(* CoDeSys 2.3.9.50 project: Indo_Tex.pro *)
(* Libraries: COMlibV2.lib 24.2.14 12:45:46, FB_DateTime.lib 15.2.16 16:36:26, TcMath.lib 23.9.04 14:15:30, SysLibVisu.lib 7.7.04 17:17:22, SysLibTargetVisu.lib 16.6.08 15:24:26, TcEtherCAT.lib 30.11.16 18:52:18, TcUtilities.lib 3.2.16 15:08:58, TcSystem.lib 7.6.16 10:01:22, TcBaseMath.lib 27.7.04 11:07:56, STANDARD.LIB 5.6.98 11:03:02, TcBase.lib 14.5.09 11:14:08, ModbusRTU.lib 19.12.16 16:50:06, TcSystemCX.lib 7.9.16 11:51:26 *)

(* Global variable list: Date_Time *)
VAR_GLOBAL
	FB_DateTime_1: FB_DateTime;
	sHourPreFix: STRING;
	sHou: STRING;
	sDayPreFix: STRING;
	sDay: STRING;
	sMonthPreFix: STRING;
	sMonth: STRING;
	sDayF: STRING;
	sMonthF: STRING;
	sDayMonth: STRING;
	sDayMonthYear: STRING;
	sDaateReport: STRING;
	sDayMonthYear1: STRING;

END_VAR

(* Global variable list: GVL_Alarm *)
VAR_GLOBAL
	RS_Error_1: RS_Error;
	RS_Error_2: RS_Error;
	RS_Error_3: RS_Error;
	RS_Error_4: RS_Error;
	RS_Error_5: RS_Error;
	RS_Error_6: RS_Error;
	RS_Error_7: RS_Error;

	bASealConvEnd1: BOOL;
	AlarmMess2: STRING(80);
	AlarmMess1: STRING(80);
	AlarWrap: STRING(80);
	CountMess: STRING(80);
	AlarmMessg: STRING(80);
	UnitASenSelet: UINT;
	SealingStep: INT;
	AlarmWrpConyMess: STRING(80);
	ConeMissAlarm: STRING(80);

	bAConeFeedCylRsError: BOOL;
	bAFwdCylRsError: BOOL;
	bAWrappingCylRsError: BOOL;
	bAWrappingCylRs1Error: BOOL;
	bAWrappingCylRs2Error: BOOL;
	bAWrappingCylRs3Error: BOOL;
	bAWrapCylRsErrorAuto: BOOL;
	bAError: BOOL;
	bASealTopCylRsError: BOOL;
	bASealBotCylRsError: BOOL;
	bASealTopBotCylRsError: BOOL;
	bASealSepXCylRsError: BOOL;
	bASealSepYCylRsError: BOOL;
	bASupplyPressureError: BOOL;
	HmiSupplyPressureMsg: STRING;
	bAFilmNotloaded: BOOL;
	bAConeMissAtSealConv: BOOL;
	bAEmergencyPressed: BOOL;
	bEmPopUp: BOOL;
	bAConeMissErrorAtWrpConv: BOOL;
	ConeAlignErr: BOOL;
	ConeMissAlarm1: STRING;
	ConeMissAlarm2: STRING;
	bAFlimNotLoaded: BOOL;
	bAPolythinSheetError: BOOL;
	bFilmErrClear: BOOL;
	bASepYAxisRsErrorChkBit: BOOL;
	bASepYAxisRsErrorChkBit1: BOOL;
	bABuzzer: BOOL;
	PressureChkTimer: TON;
	bAStop: BOOL;

	bAErrorChkBit: BOOL;
	bCheckWrappingSen: BOOL;
	bPloySheetSensError: BOOL;
	checkPolySheet2: BOOL;
	bAErrorChkBit2: BOOL;
	bCheckWrappingSen2: BOOL;
	bAErrorChkBit3: BOOL;
	bCheckWrappingSen3: BOOL;
	bWrapConvStopped2Temp: BOOL;
	SealingOk: BOOL;
	CycleComplete: BOOL;
	CycleComplete1: BOOL;
	SGrossWtNokMsg: STRING;

	SGrossWtCylEndSenErrMsg: STRING;
	bGrossWtCylEndSenError: BOOL;
END_VAR

(* Global variable list: GVL_Auto *)
VAR_GLOBAL
	bAutoModeOn: BOOL;
	bAPauseSeq: BOOL;
	bUnitBRowStopperStarted: BOOL;
	bUnitARowStopperStarted: BOOL;
	bAUnitAWeighOk: BOOL;
	bAConeFeedOver: BOOL;
	bAWrappingConvStart3: BOOL;
	bAWrappingConvStart1: BOOL;
	bAWrappingConvStart2: BOOL;
			bA3ConeWrappOver: BOOL;
	bA4thWrappOver: BOOL;
	bA6thConeWrappOver: BOOL;
	bA8thConeWrappOver: BOOL;
	bA6ConeWrappOver23: BOOL;
	AlarmMess: STRING(80);
	bAWrappingCone123OnAuto: BOOL;
	bAFwdPistonComp1: BOOL;
	bAFwdPistonComp2: BOOL;
	bAFwdPistonComp3: BOOL;
	bAConvFirstStart: BOOL;
	UnitACompleteCheckCount: CTU;
	bRetUnitAStart: BOOL;
	bRetUnitBStart: BOOL;
	bAUnitBWeighOk: BOOL;
	ConeInCompleteB: BOOL;
	(*UnitAConeCompChkCount: CTU;*)
	iSensorOnVal: USINT;
	bFwdPistonStartTemp: BOOL;
	bConeMiss1AtWrapConv: BOOL;
	bConeMiss2tWrapConv: BOOL;
	bConeMiss2AtWrapConv: BOOL;
	ConeMissbit: BOOL;
	CTU_1: CTU;
	bAPauseEnable: BOOL;
	SealComDlyTemp: TIME;
	bAMcStartInAuto: BOOL;
	bPauseExtend: BOOL;
	bAutoModeOff: BOOL;
	iTotalNoOfCones: BOOL;
	iATotalNoOfCones: INT;
	bAMcReady: BOOL;
	bAMcRunninig: BOOL;
	bAFilmLoaded: BOOL;
	bAWrapConStart: BOOL;
	bA3ConeWrappOverTemp: BOOL;
	bABypassOn: BOOL;
	bIntialAckBit: BOOL;
	ConeInComplete: BOOL;
	ConeInCompletetest: BOOL;
	ConeInCompleteTestbitB: BOOL;
	bUnitACounterDIsable: BOOL;
	ConeInCompleteA: BOOL;
	bAOneMinConvStart: BOOL;
	bAWrapwait: BOOL;
END_VAR

(* Global variable list: GVL_Hmi *)
VAR_GLOBAL
	bStopHmi: BOOL;
	bInitializeHmi: BOOL;

	HMIFeedPiston: STRING(80);
	HMIWrapPiston1: STRING(80);
	HMIWrapPiston2: STRING(80);
	HMIWrapPiston3: STRING(80);
	HMIForwdPiston:STRING(80);
	HMISealBotPiston:STRING(80);
	HMISealTopPiston:STRING(80);
	HmiXAxisPiston:STRING(80);
	HmiYAxisPiston:STRING(80);
	bErrorReset: BOOL;
	bPauseHmi: BOOL;
	bResumeHmi: BOOL;
	bResetTemp: BOOL;
	bHmiAck: BOOL;

	b18ConeModelHmi: BOOL;
	b12ConeModelHmi:BOOL;
	b24ConeModelHmi: BOOL;
	b32ConeModelHmi: BOOL;
	sAMcModeStatus: STRING;
	bAUnitBConeCrossed: BOOL;
	bAInializeStarted: BOOL;
	PopUp: BOOL;
	sAlarmStatus: STRING;
	bNegTolDisableHMI: BOOL;
	bNegTolEnableHMI: BOOL;
	bPrssurePopUp: BOOL;
	UnitAConeCountHMI: INT;
	UnitAConeCountHMI_1: INT;
	UnitBConeCountHMI: INT;
	b16ConeModelHmi: BOOL;
	WrapConeSenDetMes: STRING;
	bAmberbit2: BOOL;
	Pgm_NoHmi: INT;
	FileCreateTemp: BOOL;
	bACyclePass: BOOL;
	iCartoNoHmi: STRING;
	(*iLotNoHmi: STRING;*)
	var_1: REAL;
	var_5: REAL;
	LogYear: STRING;
	LogMonth: STRING;
	logDay: STRING;
	sTIME: STRING;
	sDATEFinal: STRING;
	DateTimeVar: STRING;
	wTodayToHmi: STRING;
	bInterlockInitial_2: BOOL;
	sMessage: STRING;
	bReadGWieght: BOOL;
	bAReset_all_error: BOOL;



	(*ProgramNoHmi:INT;
	CountCodeHmi:STRING;
	CartonNoHmi:INT;
	DefaultNetWeightHmi:REAL;
	DefaultGrossWeightHmi:REAL;
	BlendHmi:STRING;
	ShadeHmi:STRING;
	ConeTipHmi:STRING;
	ConeNettHmi:STRING;
	ConeLengthHmi:REAL;
	Cones:INT;
	Dom_ExpHmi:STRING;
	PackTypeHmi:STRING;*)




	LotASelected: BOOL;
	LotACartonNo: INT;
	LotBSelected: BOOL;
	LotBCartonNo: INT;
	LotCSelected: BOOL;
	LotDSelected: BOOL;
	LotESelected: BOOL;
	LotFSelected: BOOL;
	LotCCartonNo: INT;
	LotDCartonNo:  INT;
	LotECartonNo:  INT;
	LotFCartonNo: INT;
	LotA: INT;

	LotB: INT;

	LotC: INT;

	LotAHmi: BOOL;
	LotBHmi: BOOL;
	LotCHmi: BOOL;
	CurrentCartonNo:INT;
	LotNoChange: BOOL;
	ParametesSave: BOOL;
END_VAR

VAR_GLOBAL RETAIN
(*VAR_GLOBAL PERSISTENT*)
	b12ConeModelSelected AT %Q*: BOOL;
	b18ConeModelSelected AT %Q*: BOOL;
	b24ConeModelSelected AT %Q*: BOOL;
	b32ConeModelSelected AT %Q*: BOOL;
	rSealCompDlyHmi AT %Q*: REAL;
	iNetTolHmi AT %Q*: REAL;
	iNetWtHmi AT %Q*: REAL;
	iLotNoHmi AT %Q*: STRING;
	iWorkOrderNoHmi AT %Q*:STRING;
	NegToleranceEnabled AT %Q*: BOOL;
	b16ConeModelSelected AT %Q*: BOOL;

	ProgramNoHmi AT %Q*: INT;
	CountCodeHmi AT %Q*: STRING(80);
	CartonNoHmi AT %Q*: INT;
	DefaultNetWeightHmi AT %Q*: REAL;
	DefaultGrossWeightHmi AT %Q*: REAL;
	EmptyConeWt AT %Q*: REAL;
	BlendHmi AT %Q*: STRING(80);
	ShadeHmi AT %Q*: STRING(80);
	ConeTipHmi AT %Q*: STRING(80);
	ConeNettHmi AT %Q*: STRING(80);
	ConeLengthHmi AT %Q*: REAL;
	Cones:INT;
	Dom_ExpHmi AT %Q*: STRING(80);
	PackTypeHmi AT %Q*: STRING(80);
	ItemCodeHmi AT %Q*: STRING(80);
	IssueDesp AT %Q*: STRING(80);
	Location AT %Q*: STRING(80);
	Description AT %Q*: STRING(80);
	Remarks AT %Q*: STRING(80);
	Fyear AT %Q*: STRING(80);
	AvgCount AT %Q*: STRING(80);
	TareWeight AT %Q*: REAL;
	BarCode AT %Q*: STRING(80);
	WorkFlag AT %Q*: STRING(80);





	ItemCodeHmi1 AT %Q*: STRING(80);
	IssueDesp1 AT %Q*: STRING(80);
	Location1 AT %Q*: STRING(80);
	Description1 AT %Q*: STRING(80);
	Remarks1 AT %Q*: STRING(80);
	Fyear1 AT %Q*: STRING(80);
	AvgCount1 AT %Q*: STRING(80);
	TareWeight1 AT %Q*: REAL;
	BarCode1 AT %Q*: STRING(80);
	WorkFlag1 AT %Q*: STRING(80);
	EmptyConeWt1 AT %Q*: REAL;

	ItemCodeHmi2 AT %Q*: STRING(80);
	IssueDesp2 AT %Q*: STRING(80);
	Location2 AT %Q*: STRING(80);
	Description2 AT %Q*: STRING(80);
	Remarks2 AT %Q*: STRING(80);
	Fyear2 AT %Q*: STRING(80);
	AvgCount2 AT %Q*: STRING(80);
	TareWeight2 AT %Q*: REAL;
	BarCode2 AT %Q*: STRING(80);
	WorkFlag2 AT %Q*: STRING(80);
	EmptyConeWt2 AT %Q*: REAL;

	ItemCodeHmi3 AT %Q*: STRING(80);
	IssueDesp3 AT %Q*: STRING(80);
	Location3 AT %Q*: STRING(80);
	Description3 AT %Q*: STRING(80);
	Remarks3 AT %Q*: STRING(80);
	Fyear3 AT %Q*: STRING(80);
	AvgCount3 AT %Q*: STRING(80);
	TareWeight3 AT %Q*: REAL;
	BarCode3 AT %Q*: STRING(80);
	WorkFlag3 AT %Q*: STRING(80);
	EmptyConeWt3 AT %Q*: REAL;

	ItemCodeHmi4 AT %Q*: STRING(80);
	IssueDesp4 AT %Q*: STRING(80);
	Location4 AT %Q*: STRING(80);
	Description4 AT %Q*: STRING(80);
	Remarks4 AT %Q*: STRING(80);
	Fyear4 AT %Q*: STRING(80);
	AvgCount4 AT %Q*: STRING(80);
	TareWeight4 AT %Q*: REAL;
	BarCode4 AT %Q*: STRING(80);
	WorkFlag4 AT %Q*: STRING(80);
	EmptyConeWt4 AT %Q*: REAL;

	ItemCodeHmi5 AT %Q*: STRING(80);
	IssueDesp5 AT %Q*: STRING(80);
	Location5 AT %Q*: STRING(80);
	Description5 AT %Q*: STRING(80);
	Remarks5 AT %Q*: STRING(80);
	Fyear5 AT %Q*: STRING(80);
	AvgCount5 AT %Q*: STRING(80);
	TareWeight5 AT %Q*: REAL;
	BarCode5 AT %Q*: STRING(80);
	WorkFlag5 AT %Q*: STRING(80);
	EmptyConeWt5 AT %Q*: REAL;

	ItemCodeHmi_DIS AT %Q*: STRING(80);
	IssueDesp_DIS AT %Q*: STRING(80);
	Location_DIS AT %Q*: STRING(80);
	Description_DIS AT %Q*: STRING(80);
	Remarks_DIS AT %Q*: STRING(80);
	Fyear_DIS AT %Q*: STRING(80);
	AvgCount_DIS AT %Q*: STRING(80);
	TareWeight_DIS AT %Q*: REAL;
	BarCode_DIS AT %Q*: STRING(80);
	WorkFlag_DIS AT %Q*: STRING(80);
	EmptyConeWt_DIS AT %Q*: REAL;
END_VAR

(* Global variable list: GVL_Inputs *)
VAR_GLOBAL


(******************EL1809-1(Main)*********************)

	bIConeFeedingPistonHome AT %IX0.0: BOOL;
	bIConeFeedingPistonEnd AT %IX0.1: BOOL;
	bIConeOrientationTop AT %IX0.2: BOOL;
	bIForwardPistonHome AT %IX0.3: BOOL;
	bIForwardPistonEnd AT %IX0.4: BOOL;
	bIWrappingConeDeductionSen AT %IX0.5: BOOL;
	bISpare1 AT %IX0.6: BOOL;
	bISpare2 AT %IX0.7: BOOL;
	bISpare3 AT %IX1.0: BOOL;
	bIWrappingChannelPiston1_Home AT %IX1.1: BOOL;
	bIWrappingChannelPiston1_End AT %IX1.2: BOOL;
	bIWrappingChannelPiston2_Home AT %IX1.3: BOOL;
	bIWrappingChannelPiston2_End AT %IX1.4: BOOL;
	bIWrappingChannelPiston3_Home AT %IX1.5: BOOL;
	bIWrappingChannelPiston3_End AT %IX1.6: BOOL;
	bIWrappingCone1 AT %IX1.7:BOOL;

(******************EL1809-2(Main)*********************)

	bIWrappingCone2 AT %IX2.0: BOOL;
	bIWrappingCone3 AT %IX2.1: BOOL;
	bIWrappingFilmTensionPlate_1 AT %IX2.2: BOOL;
	bIWrappingFilmTensionPlate_2 AT %IX2.3: BOOL;
	bIWrappingFilmTensionPlate_3 AT %IX2.4: BOOL;
	bISealingTopPistonHome AT %IX2.5: BOOL;
	bISealingTopPistonEnd AT %IX2.6: BOOL;
	bISealingBottomPistonHome AT %IX2.7: BOOL;
	bISealingBottomPistonEnd AT %IX3.0: BOOL;
	bIConeCountSensor AT %IX3.1: BOOL;
	bISealingSeparatorYAxisHome AT %IX3.2: BOOL;
	bISealingSeparatorYAxisEnd AT %IX3.3: BOOL;
	bISealingSeparatorXAxisHome AT %IX3.4: BOOL;
	bISealingSeparatorXAxisEnd AT %IX3.5: BOOL;
	bIManualSealing AT %IX3.6: BOOL;
	bIPressureSwitch  AT %IX3.7: BOOL;

(******************EL1809-3(Main)*********************)

	bISpare4  AT %IX4.0: BOOL;
	bISpare5   AT %IX4.1: BOOL;
	bIUnitA_RowStopperHome   AT %IX4.2: BOOL;
	bIUnitA_RowStopperEnd AT %IX4.3: BOOL;
	bIUnitB_RowStopperHome AT %IX4.4: BOOL;
	bIUnitB_RowStopperEnd AT %IX4.5: BOOL;
	bIUnitA_StartPB AT %IX4.6: BOOL;
	bIUnitB_StartPB AT %IX4.7:BOOL;
	bIUnitAConeDetection4 AT %IX5.0:BOOL;
	bIUnitBConeDetection4 AT %IX5.1:BOOL;
	bIUnitAConeDetection1 AT %IX5.2:BOOL;
	bIUnitAConeDetection2 AT %IX5.3:BOOL;
	bIUnitAConeDetection3 AT %IX5.4:BOOL;
	bIUnitAConeCrossing AT %IX5.5:BOOL;
	bIUnitBConeDetection1 AT %IX5.6:BOOL;
	bIUnitBConeDetection2 AT %IX5.7:BOOL;

(******************EL1809-4(Main)*********************)

	bIUnitBConeDetection3 AT %IX6.0:BOOL;
	bIUnitBConeCrossing AT %IX6.1:BOOL;
	bIAutoManual AT %IX6.2:BOOL;
	bIMCStart AT %IX6.3:BOOL;
	bIMCStop AT %IX6.4:BOOL;
	bIKeySwitch AT %IX6.5:BOOL;
	bIEmergency AT %IX6.6:BOOL;
	bIUnitA_RowStopperMiddle AT %IX6.7:BOOL;

	bIUnitB_RowStopperMiddle AT %IX7.0: BOOL;
	bIGross_Crossing_Input  AT %IX7.1: BOOL;
	bIGross_Weight_Stop AT %IX7.2: BOOL;
	bIGross_Cyl_Home AT %IX7.3: BOOL;
	bIGross_Cyl_End AT %IX7.4: BOOL;
	biResetPb AT %IX7.5: BOOL;
	bISpare13 AT %IX7.6: BOOL;
	bISpare14 AT %IX7.7: BOOL;
END_VAR

(* Global variable list: GVL_Manual *)
VAR_GLOBAL




		bQMConeFeedingPistonValve :BOOL;
		bQMForwardPistonValve  :BOOL;
		bQMReversePistonValve :BOOL;
		bQMWrappingChannelPistonValve1:BOOL;
		bQMWrappingChannelPistonValve2:BOOL;
		bQMWrappingChannelPistonValve3 :BOOL;
		bQMSealingTopPistonValve :BOOL;
		bQMSealingBottomPistonValve:BOOL;


		bQMFeedingConveyorMotor :BOOL;
		bQMWrappingConveyorMotor :BOOL;
		bQMSealingConveyorMotor :BOOL;
		bQMMatrixConveyorMotor :BOOL;
		bQMFilmRollerMotor1 :BOOL;
		bQMFilmRollerMotor2 :BOOL;
		bQMFilmRollerMotor3 :BOOL;




		bQMRowStopperMotorForward  :BOOL;
		bQMRowStopperMotorReverse:BOOL;
		bQMColumnStopperMotorForward :BOOL;
		bQMColumnStopperMotorReverse:BOOL;
		bQMSealingSeparatorYAxisPistonValve :BOOL;
		bQMSealingSeparatorXAxisPistonValve :BOOL;
		bQMConeTiltingPistonValve :BOOL;
		bQMColumnPushPistonValve:BOOL;

		bQMSeparatorHorizontalPistonValveFwd :BOOL;
		bQMSeparatorVerticalPistonValve :BOOL;
		bQMCartonFeedingPistonValve :BOOL;
		bQMConeEjectionPistonValve :BOOL;
		bQMLengthTightPistonValve :BOOL;
		bQMBreadthTightPistonValve:BOOL;
		bQMEmptyCartonConveyorMotor :BOOL;
		bQMCartonConveyorMotor :BOOL;





		bQMVacuumPistonValve  :BOOL;
		bQMSeparatorHorizontalPistonValveRev  :BOOL;
		bQMSpare1  :BOOL;
		bQMSpare2 :BOOL;


	bQMUnitA_LiftPistonValve:BOOL;
	bQMUnitB_LiftPistonValve: BOOL;
	bQMUnitA_RowStopperMotorForward :BOOL;
	bQMUnitA_RowStopperMotorReverse :BOOL;
	bQMUnitB_RowStopperMotorForward :BOOL;
	bQMUnitB_RowStopperMotorReverse:BOOL;
	bQMUnitC_FullCartonConveyor :BOOL;
	bQMUnitC_LiftPistonValve :BOOL;


	bUA_LiftCylOnHmi: BOOL;
	bUA_LiftCylOffHmi: BOOL;
	bUB_LiftCylOnHmi: BOOL;
	bUB_LiftCylOffHmi: BOOL;
	bUA_RowStopperMotorFwd: BOOL;
	bUA_RowStopperMotorFwdOnHmi: BOOL;
	bUA_RowStopperMotorFwdOffHmi: BOOL;
	bUA_RowStopperMotorRevOnHmi: BOOL;
	bUB_RowStopperMotorFwdOnHmi: BOOL;
	bUB_RowStopperMotorRevOnHmi: BOOL;
	bUC_FullCartonConv: BOOL;
	bUC_FullCartonConvOnHmi: BOOL;
	bUC_FullCartonConvOffHmi: BOOL;
	bUC_LiftCylOnHmi: BOOL;
	bUC_LiftCylOffHmi: BOOL;

	bCFPistonOnHmi: BOOL;
	bCFPistonOffHmi: BOOL;
	bFPValveOnHmi:BOOL;
	bFPValveOffHmi:BOOL;
	bRPValveOnHmi:BOOL;
	bRPValveOffHmi:BOOL;
	bWrappingCPV1OnHmi:BOOL;
	bWrappingCPV1OffHmi:BOOL;
	bWrappingCPV2OnHmi:BOOL;
	bWrappingCPV2OffHmi:BOOL;
	bWrappingCPV3OnHmi:BOOL;
	bWrappingCPV3OffHmi:BOOL;
	bSealingTopPVOnHmi:BOOL;
	bSealingTopPVOffHmi:BOOL;
	bSealingBottomPVOnHmi:BOOL;
	bSealingBottomPVOffHmi:BOOL;
	bFCMotorOnHmi:BOOL;
	bFCMotorOffHmi:BOOL;
	bWCMotorOnHmi:BOOL;
	bWCMotorOffHmi:BOOL;

	bSCMotorOnHmi: BOOL;
	bSCMotorOffHmi: BOOL;
	bMCMotorOnHmi: BOOL;
	bMCMotorOffHmi: BOOL;
	bFRMotor2OnHmi: BOOL;
	bFRMotor2OffHmi: BOOL;
	bFRMotor1OnHmi: BOOL;
	bFRMotor1OffHmi: BOOL;
	bFRMotor3OnHmi: BOOL;
	bFRMotor3OffHmi: BOOL;
	bRSMotorForwardOnHmi: BOOL;
	bRSMotorForwardOffHmi: BOOL;
	bRSMotorRevOnHmi: BOOL;
	bRSMotorRevOffHmi: BOOL;
	bCSMotorFwdOnHmi: BOOL;
	bCSMotorFwdOffHmi: BOOL;
	bCSMotorRevOnHmi: BOOL;
	bCSMotorRevOffHmi: BOOL;
	bSSYAxisPistonValveOnHmi: BOOL;
	bSSYAxisPistonValveOffHmi: BOOL;
	bSSXAxisPistonValveOnHmi: BOOL;
	bSSXAxisPistonValveOffHmi: BOOL;
	bCTPistonValveOnHmi: BOOL;
	bCTPistonValveOffHmi: BOOL;
	bCPushPistonValveOnHmi: BOOL;
	bCPushPistonValveOffHmi: BOOL;
	bSHPistonValveOnHmi: BOOL;
	bSHPistonValveOffHmi: BOOL;
	bSVPistonValveOnHmi: BOOL;
	bSVPistonValveOffHmi: BOOL;
	bCPistonValveOnHmi: BOOL;
	bCPistonValveOffHmi: BOOL;
	bCEPistonValveOnHmi: BOOL;
	bCEPistonValveOffHmi: BOOL;
	bLTPistonValveOnHmi: BOOL;
	bLTPistonValveOffHmi: BOOL;
	bBTightPistonValveOnHmi: BOOL;
	bBTightPistonValveOffHmi: BOOL;
	bECCMotorOnHmi: BOOL;
	bECCMotorOffHmi: BOOL;
	bCCMotorOnHmi: BOOL;
	bCCMotorOffHmi: BOOL;
	bVPValveOnHmi: BOOL;
	bVPValveOffHmi: BOOL;
	bSHPistonValveREVOnHmi: BOOL;
	bSHPistonValveREVOffHmi: BOOL;
	bQMSeparatorHorizontalPistonValveFOR: BOOL;
	bQMColumnPushPistonValveY: BOOL;
	bCPushPistonValveYOnHmi: BOOL;
	bCPushPistonValveYOffHmi: BOOL;
	bMManualSealOn: BOOL;
	bQMLengthPistonValve: BOOL;
	bQMBreathPistonValve: BOOL;
	bQMGrossWtPiston: BOOL;
	bQMRollerConvMotor: BOOL;
	bGWPistonOffHmi1: BOOL;
	bManualModeOn: BOOL;
END_VAR

(* Global variable list: GVL_OutputFlags *)
VAR_GLOBAL



		bQAConeFeedingPistonValve  :BOOL;
		bQAForwardPistonValve  :BOOL;
		bQAWrappingChannelPistonValve1  :BOOL;
		bQAWrappingChannelPistonValve2 :BOOL;
		bQAWrappingChannelPistonValve3:BOOL;
		bQASealingTopPistonValve :BOOL;
		bQASealingBottomPistonValve:BOOL;
		bQASealingSeparatorYAxisPistonValve :BOOL;

		bQASealingSeparatorXAxisPistonValve :BOOL;
		bQAFeedingConveyorMotor :BOOL;
		bQAWrappingConveyorMotor:BOOL;
		bQAFilmRollerMotor1 :BOOL;
		bQAFilmRollerMotor2 :BOOL;
		bQAFilmRollerMotor3 :BOOL;
		bQASealingConveyorMotorFWD :BOOL;







		bQAUnitARowStopperMotorFwd  :BOOL;
		bQAUnitARowStopperMotorRev  :BOOL;
		bQAUnitBRowStopperMotorFwd  :BOOL;
		bQAUnitBRowStopperMotorRev :BOOL;
		bQAUnitAWeightOkLamp :BOOL;
		bQAUnitAWeightNokLamp  :BOOL;
		bQAUnitBWeightOkLamp :BOOL;
		bQAUnitBWeightNokLamp  :BOOL;


		bQABuzzer :BOOL;
		bQASpare1 :BOOL;
		bQASpare2 :BOOL;
		bQASpare3  :BOOL;
		bQASpare4  :BOOL;

	bQAUnitA_RowStopperMotorReverse1: BOOL;
	bQAUnitA_RowStopperMotorForward1: BOOL;
	bQASealingConveyorMotor: BOOL;

	bQASealingConveyor1: BOOL;
	bQAWrappingConveyorMotor1: BOOL;
	bQAWrappingConveyorMotor2: BOOL;
	bQAWrappingConveyorMotor3: BOOL;
	bQAAmber: BOOL;
	bQAGreen: BOOL;
	bQARed: BOOL;
	(*UnitBCompleteCheckCount: CTU;*)
END_VAR

(* Global variable list: GVL_Outputs *)
VAR_GLOBAL

		(*===============EL2809-1(Main) ===========*)


		bQConeFeedingPistonValve AT %QX0.0 :BOOL;
		bQForwardPistonValve AT %QX0.1 :BOOL;
		bQWrappingChannelPistonValve1 AT %QX0.2 :BOOL;
		bQWrappingChannelPistonValve2 AT %QX0.3:BOOL;
		bQWrappingChannelPistonValve3 AT %QX0.4:BOOL;
		bQSealingTopPistonValve AT %QX0.5:BOOL;
		bQSealingBottomPistonValve AT %QX0.6:BOOL;
		bQSealingSeparatorYAxisPistonValve AT %QX0.7:BOOL;

		bQSealingSeparatorXAxisPistonValve  AT %QX1.0:BOOL;
		bQFeedingConveyorMotor AT %QX1.1:BOOL;
		bQWrappingConveyorMotor AT %QX1.2:BOOL;
		bQFilmRollerMotor1 AT %QX1.3:BOOL;
		bQFilmRollerMotor2 AT %QX1.4:BOOL;
		bQFilmRollerMotor3 AT %QX1.5:BOOL;
		bQSealingConveyorMotorFWD AT %QX1.6:BOOL;
		bQUnitARowStopperMotorFwd AT %QX1.7:BOOL;



		(*===============EL2809-2( Main )===========*)



		bQUnitARowStopperMotorRev AT %QX2.0 :BOOL;
		bQUnitBRowStopperMotorFwd AT %QX2.1 :BOOL;
		bQUnitBRowStopperMotorRev AT %QX2.2:BOOL;
		bQUnitAWeightOkLamp  AT %QX2.3:BOOL;
		bQUnitAWeightNokLamp  AT %QX2.4:BOOL;
		bQUnitBWeightOkLamp  AT %QX2.5:BOOL;
		bQUnitBWeightNokLamp  AT %QX2.6:BOOL;
		bQTLGreen AT %QX2.7 :BOOL;

		bQTLAmber AT %QX3.0 :BOOL;
		bQTLRed AT %QX3.1 :BOOL;
		bQBuzzer AT %QX3.2 :BOOL;
		bQGross_Roller_On AT %QX3.3:BOOL;
		bQGross_Cylinder_On AT %QX3.4:BOOL;
		bQSpare3 AT %QX3.5:BOOL;
		bQSpare4  AT %QX3.6:BOOL;
		bQSpare5  AT %QX3.7:BOOL;



		(*===============EL2008-2( Main )===========*)








END_VAR

(* Global variable list: GVL_Reset *)
VAR_GLOBAL
	bQRForwardPistonValve: BOOL;
	bQRWrappingChannelPistonValve2: BOOL;
	bQRWrappingChannelPistonValve3: BOOL;
	bQRSealingTopPistonValve: BOOL;
	bQRSealingSeparatorYAxisPistonValve: BOOL;
	bQRSealingSeparatorXAxisPistonValve: BOOL;
	bQRSealingConveyorMotor: BOOL;
	bQRWrappingChannelPistonValve1: BOOL;
	bQRWrappingConveyorMotor: BOOL;
	bFwdPistonRst: BOOL;
	bARWrappingCone123OnRst: BOOL;

	bAR3ConeWrappOver: BOOL;
	bSaelUnitIntOver: BOOL;
	bWCSStart1: BOOL;
	bAInitializeSeq: BOOL;
	bSealConvIntOver: BOOL;
	sSealConvStatus: STRING;
	sWrapConvStatus: STRING;
	bWrpConvIntOver: BOOL;
	(*biResetPb: BOOL;*)
	bErrorResethmi: BOOL;

END_VAR

(* Global variable list: GVL_Serial *)
VAR_GLOBAL

	ModbusRead: BOOL;
	IADD: WORD;
	(*iNoOfRegs*)QTY: WORD;
	(*iUnitIDRead*)liD: BYTE;
	(*iBuffAddRead*)SReceiveData: ARRAY [1..5] OF BYTE;
	ModBusBussy: BOOL;
	bAModBusError: BOOL;
	rRetUnitBWeight: REAL;
	rRetUnitAWeight: REAL;
	bUnitBReadInt: BOOL;

	COMportControl: SerialLineControl;
	COMportControlError: BOOL;
	COMportControlErrorID: ComError_t;


	COMportControl_2: SerialLineControl;
	COMportControlError_2: BOOL;
	COMportControlErrorID_2: ComError_t;

	COMportControl_3: SerialLineControl;
	COMportControlError_3: BOOL;
	COMportControlErrorID_3: ComError_t;



	COMin_2_COMport_2 AT %I*: EL6inData22B;
	COMout_2_COMport_2 AT %Q*: EL6outData22B;
	TxBuffer2: ComBuffer;
	RxBuffer2: ComBuffer;

	COMin_3_COMport_3 AT %I*: EL6inData22B;
	COMout_3_COMport_3 AT %Q*: EL6outData22B;
	TxBuffer3: ComBuffer;
	RxBuffer3: ComBuffer;


	COMin_COMPort AT %I*: EL6inData22B;
	COMOut_COMPort AT %Q*: EL6outData22B;
	TxBuffer1: ComBuffer;
	RxBuffer1: ComBuffer;

	ModbusReadGross: BOOL;
	IADDGross: WORD;
	(*iNoOfRegs*)QTYGross: WORD;
	(*iUnitIDRead*)liDGross: BYTE;
	(*iBuffAddRead*)SReceiveDataGross: ARRAY [1..5] OF BYTE;
	ModBusBussyGross: BOOL;
	bAModBusErrorGross: BOOL;

	VAR_115: REAL;
	VAR_11: REAL;
	VAR_6: REAL;
	VAR_111: BYTE;
	VAR_2: BYTE;
	VAR_10: BYTE;
	VAR_12: BYTE;
	VAR_3: REAL;
	VAR_4: REAL;
	VAR_13: REAL;
	VAR_14: REAL;
	VAR_8: REAL;
	VAR_18: REAL;
	VAR_16: REAL;
	VAR_9: REAL;
	VAR_19: REAL;
	VAR_15: REAL;
	Ret_ActWt: REAL;

	VAR_115Gross: REAL;
	VAR_11Gross: REAL;
	VAR_6Gross: REAL;
	VAR_111Gross: BYTE;
	VAR_2Gross: BYTE;
	VAR_10Gross: BYTE;
	VAR_12Gross: BYTE;
	VAR_3Gross: REAL;
	VAR_4Gross: REAL;
	VAR_13Gross: REAL;
	VAR_14Gross: REAL;
	VAR_8Gross: REAL;
	VAR_18Gross: REAL;
	VAR_16Gross: REAL;
	VAR_9Gross: REAL;
	VAR_19Gross: REAL;
	VAR_15Gross: REAL;
	(*COMin_COMPort AT %I*: EL6inData22B;
	COMOut_COMPort AT %Q*: EL6outData22B;
	TxBuffer1: ComBuffer;
	RxBuffer1: ComBuffer;

	COMin_2_COMport_2 AT %I*: EL6inData22B;
	COMout_2_COMport_2 AT %Q*: EL6outData22B;
	TxBuffer2: ComBuffer;
	RxBuffer2: ComBuffer;*)

	(*COMin_3_COMport_3 AT %I*: EL6inData22B;
	COMout_3_COMport_3 AT %Q*: EL6outData22B;
	TxBuffer3: ComBuffer;
	RxBuffer3: ComBuffer;

	COMin_4_COMport_4 AT %I*: EL6inData22B;
	COMout_4_COMport_4 AT %Q*: EL6outData22B;
	TxBuffer4: ComBuffer;
	RxBuffer4: ComBuffer;*)

	rGrossWeight: REAL;
	bGrossWieghtNokTemp: BOOL;
	bGrossWieghtOk: BOOL;
	bQAGrossWieghtOkIndi: BOOL;
	bGrossWieghtNOk: BOOL;
	GrossWtReedSwBit: BOOL;
	bIGrossWtPistonHome: BOOL;
	bAGrossWtHomeSenRsError: BOOL;
	One_Min_Conv_1: INT;
	rGrossWeighToReport: REAL;
END_VAR

VAR_GLOBAL PERSISTENT
	sGrosswt AT %Q*: REAL;
	sGrossTol AT %Q*: REAL;
END_VAR

(* Global variable list: Parameters *)
VAR_GLOBAL
	SAVE: BOOL;
	TotalCones: DINT;
	iBagCount: DINT;
	LOAD: BOOL;
	PROCESSCOMPLETE: BOOL;
	sBagNoRep: STRING;
	sDayMonthYearDate: STRING;


	PRGNO_LOAD: DINT;
	NegTolEnableHmi AT %Q*: BOOL;
	NegTol1EnableHmi AT %Q*: BOOL;
	NegTol2EnableHmi AT %Q*: BOOL;
	NegTol3EnableHmi AT %Q*: BOOL;
	NegTol4EnableHmi AT %Q*: BOOL;
	NegTol5EnableHmi AT %Q*: BOOL;

	PRGNO_DIS AT %Q*: DINT;
	COUNT_DIS AT %Q*: STRING(80);
	DETAILS_DIS AT %Q*: STRING(80);
	LOTNO_DIS AT %Q*: STRING(80);
	CARTONNO_DIS AT %Q*: DINT;
	WORKORDERNO_DIS AT %Q*:STRING;
	BLEND_DIS AT %Q*:STRING;
	SHADE_DIS AT %Q*:STRING;
	CONETIP_DIS AT %Q*:STRING;
	CONELENGTH_DIS AT %Q*:REAL;
	CONENETWT_DIS AT %Q*:REAL;
	DFLTNETWT_DIS AT %Q*: REAL;
	NETWTTOL_DIS AT %Q*: REAL;
	DFLTGROSSWT_DIS AT %Q*: REAL;
	GROSSWTTOL_DIS AT %Q*: REAL;
	NegTol_DIS AT %Q*: REAL;

	negativetolerance1: BOOL;
	negativetolerance2: BOOL;
	negativetolerance3: BOOL;

	negativetolerance4: BOOL;
	negativetolerance5: BOOL;

	negativetolerance AT %Q*: BOOL;
	bABagComplete: BOOL;

	PRGNO AT %Q*: DINT;
	COUNT AT %Q*: STRING(80);
	DETAILS AT %Q*: STRING(80);
	LOTNO AT %Q*: STRING(80);
	CARTONNO AT %Q*: DINT;
	WORKORDERNO AT %Q*:STRING;
	BLEND AT %Q*:STRING;
	SHADE AT %Q*:STRING;
	CONETIP AT %Q*:STRING;
	CONELENGTH AT %Q*:REAL;
	CONENETWT AT %Q*:REAL;
	DFLTNETWT AT %Q*: REAL;
	NETWTTOL AT %Q*: REAL;
	DFLTGROSSWT AT %Q*: REAL;
	GROSSWTTOL AT %Q*: REAL;
	NegTol AT %Q*: REAL;

	PRGNO1 AT %Q*: DINT;
	COUNT1 AT %Q*: STRING(80);
	DETAILS1 AT %Q*: STRING(80);
	LOTNO1 AT %Q*: STRING(80);
	CARTONNO1 AT %Q*: DINT;
	WORKORDERNO1 AT %Q*:STRING;
	BLEND1 AT %Q*:STRING;
	SHADE1 AT %Q*:STRING;
	CONETIP1 AT %Q*:STRING;
	CONELENGTH1 AT %Q*:REAL;


	CONENETWT1 AT %Q*:REAL;
	DFLTNETWT1 AT %Q*: REAL;
	NETWTTOL1 AT %Q*: REAL;
	DFLTGROSSWT1 AT %Q*: REAL;
	GROSSWTTOL1 AT %Q*: REAL;
	NegTol1 AT %Q*: REAL;

	PRGNO2 AT %Q*: DINT;
	COUNT2 AT %Q*: STRING(80);
	DETAILS2 AT %Q*: STRING(80);
	LOTNO2 AT %Q*: STRING(80);
	CARTONNO2 AT %Q*: DINT;
	WORKORDERNO2 AT %Q*:STRING;
	BLEND2 AT %Q*:STRING;
	SHADE2 AT %Q*:STRING;
	CONETIP2 AT %Q*:STRING;
	CONELENGTH2 AT %Q*:REAL;
	CONENETWT2:REAL;
	DFLTNETWT2 AT %Q*: REAL;
	NETWTTOL2 AT %Q*: REAL;
	DFLTGROSSWT2 AT %Q*: REAL;
	GROSSWTTOL2 AT %Q*: REAL;
	NegTol2 AT %Q*: REAL;

	PRGNO3 AT %Q*: DINT;
	COUNT3 AT %Q*: STRING(80);
	DETAILS3 AT %Q*: STRING(80);
	LOTNO3 AT %Q*: STRING(80);
	CARTONNO3 AT %Q*: DINT;
	WORKORDERNO3 AT %Q*:STRING;
	BLEND3 AT %Q*:STRING;
	SHADE3 AT %Q*:STRING;
	CONETIP3 AT %Q*:STRING;
	CONELENGTH3 AT %Q*:REAL;
	CONENETWT3 AT %Q*:REAL;
	DFLTNETWT3 AT %Q*: REAL;
	NETWTTOL3 AT %Q*: REAL;
	DFLTGROSSWT3 AT %Q*: REAL;
	GROSSWTTOL3 AT %Q*: REAL;
	NegTol3 AT %Q*: REAL;

	PRGNO4 AT %Q*: DINT;
	COUNT4 AT %Q*: STRING(80);
	DETAILS4 AT %Q*: STRING(80);
	LOTNO4 AT %Q*: STRING(80);
	CARTONNO4 AT %Q*: DINT;
	WORKORDERNO4 AT %Q*:STRING;
	BLEND4 AT %Q*:STRING;
	SHADE4 AT %Q*:STRING;
	CONETIP4 AT %Q*:STRING;
	CONELENGTH4 AT %Q*:REAL;
	CONENETWT4:REAL;
	DFLTNETWT4 AT %Q*: REAL;
	NETWTTOL4 AT %Q*: REAL;
	DFLTGROSSWT4 AT %Q*: REAL;
	GROSSWTTOL4 AT %Q*: REAL;
	NegTol4 AT %Q*: REAL;


	PRGNO5 AT %Q*: DINT;
	COUNT5 AT %Q*: STRING(80);
	DETAILS5 AT %Q*: STRING(80);
	LOTNO5 AT %Q*: STRING(80);
	CARTONNO5 AT %Q*: DINT;
	WORKORDERNO5 AT %Q*:STRING;
	BLEND5 AT %Q*:STRING;
	SHADE5 AT %Q*:STRING;
	CONETIP5 AT %Q*:STRING;
	CONELENGTH5 AT %Q*:REAL;
	CONENETWT5 AT %Q*:REAL;
	DFLTNETWT5 AT %Q*: REAL;
	NETWTTOL5 AT %Q*: REAL;
	DFLTGROSSWT5 AT %Q*: REAL;
	GROSSWTTOL5 AT %Q*: REAL;
	NegTol5 AT %Q*: REAL;

	DOM_EXPORT AT %Q*: STRING;
	PACKTYPE AT %Q*: STRING;
	DOM_EXPORT1 AT %Q*: STRING;
	PACKTYPE1 AT %Q*: STRING;
	DOM_EXPORT2 AT %Q*: STRING;
	PACKTYPE2 AT %Q*: STRING;
	DOM_EXPORT3 AT %Q*: STRING;
	PACKTYPE3 AT %Q*: STRING;
	DOM_EXPORT4 AT %Q*: STRING;
	PACKTYPE4 AT %Q*: STRING;
	DOM_EXPORT5 AT %Q*: STRING;
	DOM_EXPORT_DIS AT %Q*: STRING;
	PACKTYPE5 AT %Q*: STRING;
	PACKTYPE_DIS AT %Q*: STRING;

	NOOFCONES: DINT;
	NOOFCONES1: DINT;
	NOOFCONES2: DINT;
	NOOFCONES3: DINT;
	NOOFCONES4: DINT;
	NOOFCONES5: DINT;
	NOOFCONES_DIS: DINT;



	PRGNO6:DINT;
	COUNT6:STRING;
	DETAILS6:STRING;
	LOTNO6:STRING;
	CARTONNO6:DINT;
	WORKORDERNO6:STRING;
	BLEND6:STRING;
	SHADE6:STRING;
	CONETIP6:STRING;
	CONELENGTH6:REAL;
	CONENETWT6:REAL;
	DFLTNETWT6:REAL;
	NETWTTOL6:REAL;
	DFLTGROSSWT6:REAL;
	GROSSWTTOL6:REAL;


	PRGNO7:DINT;
	COUNT7:STRING;
	DETAILS7:STRING;
	LOTNO7:STRING;
	CARTONNO7:DINT;
	WORKORDERNO7:STRING;
	BLEND7:STRING;
	SHADE7:STRING;
	CONETIP7:STRING;
	CONELENGTH7:REAL;
	CONENETWT7:REAL;
	DFLTNETWT7:REAL;
	NETWTTOL7:REAL;
	DFLTGROSSWT7:REAL;
	GROSSWTTOL7:REAL;


	PRGNO8:DINT;
	COUNT8:STRING;
	DETAILS8:STRING;
	LOTNO8:STRING;
	CARTONNO8:DINT;
	WORKORDERNO8:STRING;
	BLEND8:STRING;
	SHADE8:STRING;
	CONETIP8:STRING;
	CONELENGTH8:REAL;
	CONENETWT8:REAL;
	DFLTNETWT8:REAL;
	NETWTTOL8:REAL;
	DFLTGROSSWT8:REAL;
	GROSSWTTOL8:REAL;


	PRGNO9:DINT;
	COUNT9:STRING;
	DETAILS9:STRING;
	LOTNO9:STRING;
	CARTONNO9:DINT;
	WORKORDERNO9:STRING;
	BLEND9:STRING;
	SHADE9:STRING;
	CONETIP9:STRING;
	CONELENGTH9:REAL;
	CONENETWT9:REAL;
	DFLTNETWT9:REAL;
	NETWTTOL9:REAL;
	DFLTGROSSWT9:REAL;
	GROSSWTTOL9:REAL;


	PRGNO10:DINT;
	COUNT10:STRING;
	DETAILS10:STRING;
	LOTNO10:STRING;
	CARTONNO10:DINT;
	WORKORDERNO10:STRING;
	BLEND10:STRING;
	SHADE10:STRING;
	CONETIP10:STRING;
	CONELENGTH10:REAL;
	CONENETWT10:REAL;
	DFLTNETWT10:REAL;
	NETWTTOL10:REAL;
	DFLTGROSSWT10:REAL;
	GROSSWTTOL10:REAL;

	PRG1RUNNING AT %Q*: BOOL;
	PRG2RUNNING AT %Q*: BOOL;
	PRG3RUNNING AT %Q*: BOOL;
	PRG4RUNNING AT %Q*: BOOL;
	PRG5RUNNING AT %Q*: BOOL;
	PRG6RUNNING: BOOL;
	PRG7RUNNING: BOOL;
	PRG8RUNNING: BOOL;
	PRG9RUNNING: BOOL;
	PRG10RUNNING: BOOL;
	PRINTENABLE: BOOL;
	PRINTENABLED: BOOL;

	DfltWtPrint: BOOL;
	DfltGrossWtPrint_En: BOOL;
	GrossWtPrintDflt: BOOL;
	NetwtPrint: STRING;
	GrosswtPrint: STRING;

	ReportPath: STRING;
	sDayF1: STRING;
	sMonthF1: STRING;
	sDayMonth1: STRING;

	ReportPath_Final_2: STRING;
	FB_DateTime_2: FB_DateTime;











	ReportPath_Final_1: STRING;
	ReportPath_Final: STRING;


END_VAR

(* Global variable list: Print *)
VAR_GLOBAL
	(*FileCreateTemp: BOOL;*)
	ProductionData_Print: STRING(255);
	ProductionDataValues_Print: STRING(255);
	ProductionDataValues_Print_Com:STRING(255);
	PrintOk: BOOL;
	PrintEnableHmi: BOOL;
	PrintValue: INT;
	bANewDay: BOOL;
	ProductionDataValues_IndoPrint: STRING(255);
	ProductionData_IndoPrint: STRING(255);
	ProductionDataError_IndoPrint: STRING(255);

	ProductionData_IndoPrint2:STRING(255);
	ProductionDataError_IndoPrint2:STRING(255);
	ProductionDataValues_IndoPrint_Com:STRING(255);
		ProductionDataValuesError_IndoPrint_Com:STRING(255);
	ProductionData_IndoPrint11 : ProductionData_IndoPrint1;
	ProductionData_IndoPrintError11 : ProductionDataError_IndoPrint1;


	ReportPrint:BOOL;




	ReportPathError: STRING;
	ReportPath_FinalError: STRING;
	ReportPath_Final_1Error: STRING;
	ReportPath_Final_2Error: STRING;

	SerialNo AT %Q*: DINT;
	BagSerialNo: DINT;

	ReportSave: BOOL;
	SerialNoError: DINT;




	Default_GrossWeight_Report: STRING;
	Actual_NetWeight_Report: STRING;
	Actual_GrossWeight_Report: STRING;
	ActualNetWeight: REAL;
	ActualGrossWeight: REAL;
	Default_NetWeight_Report: STRING;
	DefaultNetWt AT %Q*: REAL;
	NetWtTolRep AT %Q*: REAL;
	DefaultGrossWt AT %Q*: REAL;
	GrossWtTolRep AT %Q*: REAL;

END_VAR

(* Global variable list: TwinCAT_Configuration *)
(* Generated automatically by TwinCAT - (read only) *)
VAR_CONFIG
	Serial.ModbusRtuMaster_KL6x22B_3.InData AT %IB8 : MB_KL6inData22B;
	Serial.ModbusRtuMaster_KL6x22B_3.OutData AT %QB5752 : MB_KL6outData22B;
	Serial.ModbusRtuMaster_KL6x22B_4.InData AT %IB32 : MB_KL6inData22B;
	Serial.ModbusRtuMaster_KL6x22B_4.OutData AT %QB5776 : MB_KL6outData22B;
	.b12ConeModelSelected AT %QX5748.0 : BOOL;	(*  ~ {LinkedWith:TIID^Device 3 (NOV/DP-RAM)^Outputs^Var 570} *)
	.b18ConeModelSelected AT %QX5748.1 : BOOL;	(*  ~ {LinkedWith:TIID^Device 3 (NOV/DP-RAM)^Outputs^Var 571} *)
	.b24ConeModelSelected AT %QX5748.2 : BOOL;	(*  ~ {LinkedWith:TIID^Device 3 (NOV/DP-RAM)^Outputs^Var 572} *)
	.b32ConeModelSelected AT %QX5748.3 : BOOL;	(*  ~ {LinkedWith:TIID^Device 3 (NOV/DP-RAM)^Outputs^Var 573} *)
	.rSealCompDlyHmi AT %QB4 : REAL;	(*  ~ {LinkedWith:TIID^Device 3 (NOV/DP-RAM)^Outputs^Var 576} *)
	.iNetTolHmi AT %QB8 : REAL;	(*  ~ {LinkedWith:TIID^Device 3 (NOV/DP-RAM)^Outputs^Var 577} *)
	.iNetWtHmi AT %QB12 : REAL;	(*  ~ {LinkedWith:TIID^Device 3 (NOV/DP-RAM)^Outputs^Var 578} *)
	.iLotNoHmi AT %QB16 : STRING(80);
	.iWorkOrderNoHmi AT %QB100 : STRING(80);
	.NegToleranceEnabled AT %QX5748.4 : BOOL;	(*  ~ {LinkedWith:TIID^Device 3 (NOV/DP-RAM)^Outputs^Var 574} *)
	.b16ConeModelSelected AT %QX5748.5 : BOOL;	(*  ~ {LinkedWith:TIID^Device 3 (NOV/DP-RAM)^Outputs^Var 575} *)
	.ProgramNoHmi AT %QB5800 : INT;
	.CountCodeHmi AT %QB5804 : STRING(80);
	.CartonNoHmi AT %QB5886 : INT;
	.DefaultNetWeightHmi AT %QB5888 : REAL;
	.DefaultGrossWeightHmi AT %QB5892 : REAL;
	.EmptyConeWt AT %QB5896 : REAL;
	.BlendHmi AT %QB5900 : STRING(80);
	.ShadeHmi AT %QB5984 : STRING(80);
	.ConeTipHmi AT %QB6068 : STRING(80);
	.ConeNettHmi AT %QB6152 : STRING(80);
	.ConeLengthHmi AT %QB6236 : REAL;
	.Dom_ExpHmi AT %QB6240 : STRING(80);
	.PackTypeHmi AT %QB6324 : STRING(80);
	.ItemCodeHmi AT %QB6408 : STRING(80);
	.IssueDesp AT %QB6492 : STRING(80);
	.Location AT %QB6576 : STRING(80);
	.Description AT %QB6660 : STRING(80);
	.Remarks AT %QB6744 : STRING(80);
	.Fyear AT %QB6828 : STRING(80);
	.AvgCount AT %QB6912 : STRING(80);
	.TareWeight AT %QB6996 : REAL;
	.BarCode AT %QB7000 : STRING(80);
	.WorkFlag AT %QB7084 : STRING(80);
	.ItemCodeHmi1 AT %QB7168 : STRING(80);	(*  ~ {LinkedWith:TIID^Device 3 (NOV/DP-RAM)^Outputs^Var 719} *)
	.IssueDesp1 AT %QB7252 : STRING(80);	(*  ~ {LinkedWith:TIID^Device 3 (NOV/DP-RAM)^Outputs^Var 718} *)
	.Location1 AT %QB7336 : STRING(80);	(*  ~ {LinkedWith:TIID^Device 3 (NOV/DP-RAM)^Outputs^Var 717} *)
	.Description1 AT %QB7420 : STRING(80);	(*  ~ {LinkedWith:TIID^Device 3 (NOV/DP-RAM)^Outputs^Var 716} *)
	.Remarks1 AT %QB7504 : STRING(80);	(*  ~ {LinkedWith:TIID^Device 3 (NOV/DP-RAM)^Outputs^Var 715} *)
	.Fyear1 AT %QB7588 : STRING(80);	(*  ~ {LinkedWith:TIID^Device 3 (NOV/DP-RAM)^Outputs^Var 714} *)
	.AvgCount1 AT %QB7672 : STRING(80);	(*  ~ {LinkedWith:TIID^Device 3 (NOV/DP-RAM)^Outputs^Var 713} *)
	.TareWeight1 AT %QB7756 : REAL;
	.BarCode1 AT %QB7760 : STRING(80);	(*  ~ {LinkedWith:TIID^Device 3 (NOV/DP-RAM)^Outputs^Var 712} *)
	.WorkFlag1 AT %QB7844 : STRING(80);	(*  ~ {LinkedWith:TIID^Device 3 (NOV/DP-RAM)^Outputs^Var 711} *)
	.EmptyConeWt1 AT %QB7928 : REAL;
	.ItemCodeHmi2 AT %QB7932 : STRING(80);	(*  ~ {LinkedWith:TIID^Device 3 (NOV/DP-RAM)^Outputs^Var 710} *)
	.IssueDesp2 AT %QB8016 : STRING(80);	(*  ~ {LinkedWith:TIID^Device 3 (NOV/DP-RAM)^Outputs^Var 709} *)
	.Location2 AT %QB8100 : STRING(80);	(*  ~ {LinkedWith:TIID^Device 3 (NOV/DP-RAM)^Outputs^Var 708} *)
	.Description2 AT %QB8184 : STRING(80);	(*  ~ {LinkedWith:TIID^Device 3 (NOV/DP-RAM)^Outputs^Var 707} *)
	.Remarks2 AT %QB8268 : STRING(80);	(*  ~ {LinkedWith:TIID^Device 3 (NOV/DP-RAM)^Outputs^Var 706} *)
	.Fyear2 AT %QB8352 : STRING(80);	(*  ~ {LinkedWith:TIID^Device 3 (NOV/DP-RAM)^Outputs^Var 705} *)
	.AvgCount2 AT %QB8436 : STRING(80);	(*  ~ {LinkedWith:TIID^Device 3 (NOV/DP-RAM)^Outputs^Var 704} *)
	.TareWeight2 AT %QB8520 : REAL;
	.BarCode2 AT %QB8524 : STRING(80);	(*  ~ {LinkedWith:TIID^Device 3 (NOV/DP-RAM)^Outputs^Var 703} *)
	.WorkFlag2 AT %QB8608 : STRING(80);	(*  ~ {LinkedWith:TIID^Device 3 (NOV/DP-RAM)^Outputs^Var 702} *)
	.EmptyConeWt2 AT %QB8692 : REAL;
	.ItemCodeHmi3 AT %QB8696 : STRING(80);	(*  ~ {LinkedWith:TIID^Device 3 (NOV/DP-RAM)^Outputs^Var 701} *)
	.IssueDesp3 AT %QB8780 : STRING(80);	(*  ~ {LinkedWith:TIID^Device 3 (NOV/DP-RAM)^Outputs^Var 700} *)
	.Location3 AT %QB8864 : STRING(80);	(*  ~ {LinkedWith:TIID^Device 3 (NOV/DP-RAM)^Outputs^Var 699} *)
	.Description3 AT %QB8948 : STRING(80);	(*  ~ {LinkedWith:TIID^Device 3 (NOV/DP-RAM)^Outputs^Var 698} *)
	.Remarks3 AT %QB9032 : STRING(80);	(*  ~ {LinkedWith:TIID^Device 3 (NOV/DP-RAM)^Outputs^Var 697} *)
	.Fyear3 AT %QB9116 : STRING(80);	(*  ~ {LinkedWith:TIID^Device 3 (NOV/DP-RAM)^Outputs^Var 684} *)
	.AvgCount3 AT %QB9200 : STRING(80);	(*  ~ {LinkedWith:TIID^Device 3 (NOV/DP-RAM)^Outputs^Var 683} *)
	.TareWeight3 AT %QB9284 : REAL;
	.BarCode3 AT %QB9288 : STRING(80);	(*  ~ {LinkedWith:TIID^Device 3 (NOV/DP-RAM)^Outputs^Var 682} *)
	.WorkFlag3 AT %QB9372 : STRING(80);	(*  ~ {LinkedWith:TIID^Device 3 (NOV/DP-RAM)^Outputs^Var 681} *)
	.EmptyConeWt3 AT %QB9456 : REAL;
	.ItemCodeHmi4 AT %QB9460 : STRING(80);	(*  ~ {LinkedWith:TIID^Device 3 (NOV/DP-RAM)^Outputs^Var 680} *)
	.IssueDesp4 AT %QB9544 : STRING(80);	(*  ~ {LinkedWith:TIID^Device 3 (NOV/DP-RAM)^Outputs^Var 679} *)
	.Location4 AT %QB9628 : STRING(80);	(*  ~ {LinkedWith:TIID^Device 3 (NOV/DP-RAM)^Outputs^Var 678} *)
	.Description4 AT %QB9712 : STRING(80);	(*  ~ {LinkedWith:TIID^Device 3 (NOV/DP-RAM)^Outputs^Var 677} *)
	.Remarks4 AT %QB9796 : STRING(80);	(*  ~ {LinkedWith:TIID^Device 3 (NOV/DP-RAM)^Outputs^Var 676} *)
	.Fyear4 AT %QB9880 : STRING(80);	(*  ~ {LinkedWith:TIID^Device 3 (NOV/DP-RAM)^Outputs^Var 675} *)
	.AvgCount4 AT %QB9964 : STRING(80);	(*  ~ {LinkedWith:TIID^Device 3 (NOV/DP-RAM)^Outputs^Var 674} *)
	.TareWeight4 AT %QB10048 : REAL;
	.BarCode4 AT %QB10052 : STRING(80);	(*  ~ {LinkedWith:TIID^Device 3 (NOV/DP-RAM)^Outputs^Var 673} *)
	.WorkFlag4 AT %QB10136 : STRING(80);	(*  ~ {LinkedWith:TIID^Device 3 (NOV/DP-RAM)^Outputs^Var 672} *)
	.EmptyConeWt4 AT %QB10220 : REAL;
	.ItemCodeHmi5 AT %QB10224 : STRING(80);	(*  ~ {LinkedWith:TIID^Device 3 (NOV/DP-RAM)^Outputs^Var 671} *)
	.IssueDesp5 AT %QB10308 : STRING(80);	(*  ~ {LinkedWith:TIID^Device 3 (NOV/DP-RAM)^Outputs^Var 670} *)
	.Location5 AT %QB10392 : STRING(80);	(*  ~ {LinkedWith:TIID^Device 3 (NOV/DP-RAM)^Outputs^Var 669} *)
	.Description5 AT %QB10476 : STRING(80);	(*  ~ {LinkedWith:TIID^Device 3 (NOV/DP-RAM)^Outputs^Var 668} *)
	.Remarks5 AT %QB10560 : STRING(80);	(*  ~ {LinkedWith:TIID^Device 3 (NOV/DP-RAM)^Outputs^Var 667} *)
	.Fyear5 AT %QB10644 : STRING(80);	(*  ~ {LinkedWith:TIID^Device 3 (NOV/DP-RAM)^Outputs^Var 666} *)
	.AvgCount5 AT %QB10728 : STRING(80);	(*  ~ {LinkedWith:TIID^Device 3 (NOV/DP-RAM)^Outputs^Var 665} *)
	.TareWeight5 AT %QB10812 : REAL;
	.BarCode5 AT %QB10816 : STRING(80);	(*  ~ {LinkedWith:TIID^Device 3 (NOV/DP-RAM)^Outputs^Var 664} *)
	.WorkFlag5 AT %QB10900 : STRING(80);	(*  ~ {LinkedWith:TIID^Device 3 (NOV/DP-RAM)^Outputs^Var 663} *)
	.EmptyConeWt5 AT %QB10984 : REAL;
	.ItemCodeHmi_DIS AT %QB10988 : STRING(80);	(*  ~ {LinkedWith:TIID^Device 3 (NOV/DP-RAM)^Outputs^Var 662} *)
	.IssueDesp_DIS AT %QB11072 : STRING(80);	(*  ~ {LinkedWith:TIID^Device 3 (NOV/DP-RAM)^Outputs^Var 661} *)
	.Location_DIS AT %QB11156 : STRING(80);	(*  ~ {LinkedWith:TIID^Device 3 (NOV/DP-RAM)^Outputs^Var 660} *)
	.Description_DIS AT %QB11240 : STRING(80);	(*  ~ {LinkedWith:TIID^Device 3 (NOV/DP-RAM)^Outputs^Var 659} *)
	.Remarks_DIS AT %QB11324 : STRING(80);	(*  ~ {LinkedWith:TIID^Device 3 (NOV/DP-RAM)^Outputs^Var 658} *)
	.Fyear_DIS AT %QB11408 : STRING(80);	(*  ~ {LinkedWith:TIID^Device 3 (NOV/DP-RAM)^Outputs^Var 657} *)
	.AvgCount_DIS AT %QB11492 : STRING(80);	(*  ~ {LinkedWith:TIID^Device 3 (NOV/DP-RAM)^Outputs^Var 656} *)
	.TareWeight_DIS AT %QB11576 : REAL;
	.BarCode_DIS AT %QB11580 : STRING(80);	(*  ~ {LinkedWith:TIID^Device 3 (NOV/DP-RAM)^Outputs^Var 655} *)
	.WorkFlag_DIS AT %QB11664 : STRING(80);	(*  ~ {LinkedWith:TIID^Device 3 (NOV/DP-RAM)^Outputs^Var 654} *)
	.EmptyConeWt_DIS AT %QB11748 : REAL;
	.COMin_2_COMport_2 AT %IB56 : EL6inData22B;
	.COMout_2_COMport_2 AT %QB11752 : EL6outData22B;
	.COMin_3_COMport_3 AT %IB80 : EL6inData22B;
	.COMout_3_COMport_3 AT %QB11776 : EL6outData22B;
	.COMin_COMPort AT %IB104 : EL6inData22B;
	.COMOut_COMPort AT %QB11800 : EL6outData22B;
	.sGrosswt AT %QB184 : REAL;	(*  ~ {LinkedWith:TIID^Device 3 (NOV/DP-RAM)^Outputs^Var 579} *)
	.sGrossTol AT %QB188 : REAL;	(*  ~ {LinkedWith:TIID^Device 3 (NOV/DP-RAM)^Outputs^Var 580} *)
	.NegTolEnableHmi AT %QX5748.6 : BOOL;	(*  ~ {LinkedWith:TIID^Device 3 (NOV/DP-RAM)^Outputs^Var 723} *)
	.NegTol1EnableHmi AT %QX5748.7 : BOOL;	(*  ~ {LinkedWith:TIID^Device 3 (NOV/DP-RAM)^Outputs^Var 724} *)
	.NegTol2EnableHmi AT %QX5749.0 : BOOL;	(*  ~ {LinkedWith:TIID^Device 3 (NOV/DP-RAM)^Outputs^Var 725} *)
	.NegTol3EnableHmi AT %QX5749.1 : BOOL;	(*  ~ {LinkedWith:TIID^Device 3 (NOV/DP-RAM)^Outputs^Var 726} *)
	.NegTol4EnableHmi AT %QX5749.2 : BOOL;	(*  ~ {LinkedWith:TIID^Device 3 (NOV/DP-RAM)^Outputs^Var 727} *)
	.NegTol5EnableHmi AT %QX5749.3 : BOOL;	(*  ~ {LinkedWith:TIID^Device 3 (NOV/DP-RAM)^Outputs^Var 728} *)
	.PRGNO_DIS AT %QB192 : DINT;	(*  ~ {LinkedWith:TIID^Device 3 (NOV/DP-RAM)^Outputs^Var 267} *)
	.COUNT_DIS AT %QB196 : STRING(80);	(*  ~ {LinkedWith:TIID^Device 3 (NOV/DP-RAM)^Outputs^Var 261} *)
	.DETAILS_DIS AT %QB280 : STRING(80);
	.LOTNO_DIS AT %QB364 : STRING(80);	(*  ~ {LinkedWith:TIID^Device 3 (NOV/DP-RAM)^Outputs^Var 268} *)
	.CARTONNO_DIS AT %QB448 : DINT;	(*  ~ {LinkedWith:TIID^Device 3 (NOV/DP-RAM)^Outputs^Var 315} *)
	.WORKORDERNO_DIS AT %QB452 : STRING(80);	(*  ~ {LinkedWith:TIID^Device 3 (NOV/DP-RAM)^Outputs^Var 274} *)
	.BLEND_DIS AT %QB536 : STRING(80);	(*  ~ {LinkedWith:TIID^Device 3 (NOV/DP-RAM)^Outputs^Var 280} *)
	.SHADE_DIS AT %QB620 : STRING(80);	(*  ~ {LinkedWith:TIID^Device 3 (NOV/DP-RAM)^Outputs^Var 286} *)
	.CONETIP_DIS AT %QB704 : STRING(80);	(*  ~ {LinkedWith:TIID^Device 3 (NOV/DP-RAM)^Outputs^Var 292} *)
	.CONELENGTH_DIS AT %QB788 : REAL;	(*  ~ {LinkedWith:TIID^Device 3 (NOV/DP-RAM)^Outputs^Var 321} *)
	.CONENETWT_DIS AT %QB792 : REAL;	(*  ~ {LinkedWith:TIID^Device 3 (NOV/DP-RAM)^Outputs^Var 323} *)
	.DFLTNETWT_DIS AT %QB796 : REAL;	(*  ~ {LinkedWith:TIID^Device 3 (NOV/DP-RAM)^Outputs^Var 332} *)
	.NETWTTOL_DIS AT %QB800 : REAL;	(*  ~ {LinkedWith:TIID^Device 3 (NOV/DP-RAM)^Outputs^Var 333} *)
	.DFLTGROSSWT_DIS AT %QB804 : REAL;	(*  ~ {LinkedWith:TIID^Device 3 (NOV/DP-RAM)^Outputs^Var 334} *)
	.GROSSWTTOL_DIS AT %QB808 : REAL;	(*  ~ {LinkedWith:TIID^Device 3 (NOV/DP-RAM)^Outputs^Var 335} *)
	.NegTol_DIS AT %QB812 : REAL;	(*  ~ {LinkedWith:TIID^Device 3 (NOV/DP-RAM)^Outputs^Var 356} *)
	.negativetolerance AT %QX5749.4 : BOOL;	(*  ~ {LinkedWith:TIID^Device 3 (NOV/DP-RAM)^Outputs^Var 729} *)
	.PRGNO AT %QB816 : DINT;
	.COUNT AT %QB820 : STRING(80);
	.DETAILS AT %QB904 : STRING(80);
	.LOTNO AT %QB988 : STRING(80);
	.CARTONNO AT %QB1072 : DINT;
	.WORKORDERNO AT %QB1076 : STRING(80);
	.BLEND AT %QB1160 : STRING(80);
	.SHADE AT %QB1244 : STRING(80);
	.CONETIP AT %QB1328 : STRING(80);
	.CONELENGTH AT %QB1412 : REAL;
	.CONENETWT AT %QB1416 : REAL;
	.DFLTNETWT AT %QB1420 : REAL;
	.NETWTTOL AT %QB1424 : REAL;
	.DFLTGROSSWT AT %QB1428 : REAL;
	.GROSSWTTOL AT %QB1432 : REAL;
	.NegTol AT %QB1436 : REAL;
	.PRGNO1 AT %QB1440 : DINT;	(*  ~ {LinkedWith:TIID^Device 3 (NOV/DP-RAM)^Outputs^Var 310} *)
	.COUNT1 AT %QB1444 : STRING(80);	(*  ~ {LinkedWith:TIID^Device 3 (NOV/DP-RAM)^Outputs^Var 262} *)
	.DETAILS1 AT %QB1528 : STRING(80);
	.LOTNO1 AT %QB1612 : STRING(80);	(*  ~ {LinkedWith:TIID^Device 3 (NOV/DP-RAM)^Outputs^Var 269} *)
	.CARTONNO1 AT %QB1696 : DINT;	(*  ~ {LinkedWith:TIID^Device 3 (NOV/DP-RAM)^Outputs^Var 316} *)
	.WORKORDERNO1 AT %QB1700 : STRING(80);	(*  ~ {LinkedWith:TIID^Device 3 (NOV/DP-RAM)^Outputs^Var 275} *)
	.BLEND1 AT %QB1784 : STRING(80);	(*  ~ {LinkedWith:TIID^Device 3 (NOV/DP-RAM)^Outputs^Var 281} *)
	.SHADE1 AT %QB1868 : STRING(80);	(*  ~ {LinkedWith:TIID^Device 3 (NOV/DP-RAM)^Outputs^Var 287} *)
	.CONETIP1 AT %QB1952 : STRING(80);	(*  ~ {LinkedWith:TIID^Device 3 (NOV/DP-RAM)^Outputs^Var 293} *)
	.CONELENGTH1 AT %QB2036 : REAL;	(*  ~ {LinkedWith:TIID^Device 3 (NOV/DP-RAM)^Outputs^Var 324} *)
	.CONENETWT1 AT %QB2040 : REAL;	(*  ~ {LinkedWith:TIID^Device 3 (NOV/DP-RAM)^Outputs^Var 325} *)
	.DFLTNETWT1 AT %QB2044 : REAL;	(*  ~ {LinkedWith:TIID^Device 3 (NOV/DP-RAM)^Outputs^Var 336} *)
	.NETWTTOL1 AT %QB2048 : REAL;	(*  ~ {LinkedWith:TIID^Device 3 (NOV/DP-RAM)^Outputs^Var 337} *)
	.DFLTGROSSWT1 AT %QB2052 : REAL;	(*  ~ {LinkedWith:TIID^Device 3 (NOV/DP-RAM)^Outputs^Var 338} *)
	.GROSSWTTOL1 AT %QB2056 : REAL;	(*  ~ {LinkedWith:TIID^Device 3 (NOV/DP-RAM)^Outputs^Var 339} *)
	.NegTol1 AT %QB2060 : REAL;
	.PRGNO2 AT %QB2064 : DINT;	(*  ~ {LinkedWith:TIID^Device 3 (NOV/DP-RAM)^Outputs^Var 311} *)
	.COUNT2 AT %QB2068 : STRING(80);	(*  ~ {LinkedWith:TIID^Device 3 (NOV/DP-RAM)^Outputs^Var 263} *)
	.DETAILS2 AT %QB2152 : STRING(80);
	.LOTNO2 AT %QB2236 : STRING(80);	(*  ~ {LinkedWith:TIID^Device 3 (NOV/DP-RAM)^Outputs^Var 270} *)
	.CARTONNO2 AT %QB2320 : DINT;	(*  ~ {LinkedWith:TIID^Device 3 (NOV/DP-RAM)^Outputs^Var 317} *)
	.WORKORDERNO2 AT %QB2324 : STRING(80);	(*  ~ {LinkedWith:TIID^Device 3 (NOV/DP-RAM)^Outputs^Var 276} *)
	.BLEND2 AT %QB2408 : STRING(80);	(*  ~ {LinkedWith:TIID^Device 3 (NOV/DP-RAM)^Outputs^Var 282} *)
	.SHADE2 AT %QB2492 : STRING(80);	(*  ~ {LinkedWith:TIID^Device 3 (NOV/DP-RAM)^Outputs^Var 288} *)
	.CONETIP2 AT %QB2576 : STRING(80);	(*  ~ {LinkedWith:TIID^Device 3 (NOV/DP-RAM)^Outputs^Var 294} *)
	.CONELENGTH2 AT %QB2660 : REAL;	(*  ~ {LinkedWith:TIID^Device 3 (NOV/DP-RAM)^Outputs^Var 326} *)
	.DFLTNETWT2 AT %QB2664 : REAL;	(*  ~ {LinkedWith:TIID^Device 3 (NOV/DP-RAM)^Outputs^Var 340} *)
	.NETWTTOL2 AT %QB2668 : REAL;	(*  ~ {LinkedWith:TIID^Device 3 (NOV/DP-RAM)^Outputs^Var 341} *)
	.DFLTGROSSWT2 AT %QB2672 : REAL;	(*  ~ {LinkedWith:TIID^Device 3 (NOV/DP-RAM)^Outputs^Var 342} *)
	.GROSSWTTOL2 AT %QB2676 : REAL;	(*  ~ {LinkedWith:TIID^Device 3 (NOV/DP-RAM)^Outputs^Var 343} *)
	.NegTol2 AT %QB2680 : REAL;
	.PRGNO3 AT %QB2684 : DINT;	(*  ~ {LinkedWith:TIID^Device 3 (NOV/DP-RAM)^Outputs^Var 312} *)
	.COUNT3 AT %QB2688 : STRING(80);	(*  ~ {LinkedWith:TIID^Device 3 (NOV/DP-RAM)^Outputs^Var 264} *)
	.DETAILS3 AT %QB2772 : STRING(80);
	.LOTNO3 AT %QB2856 : STRING(80);	(*  ~ {LinkedWith:TIID^Device 3 (NOV/DP-RAM)^Outputs^Var 271} *)
	.CARTONNO3 AT %QB2940 : DINT;	(*  ~ {LinkedWith:TIID^Device 3 (NOV/DP-RAM)^Outputs^Var 318} *)
	.WORKORDERNO3 AT %QB2944 : STRING(80);	(*  ~ {LinkedWith:TIID^Device 3 (NOV/DP-RAM)^Outputs^Var 277} *)
	.BLEND3 AT %QB3028 : STRING(80);	(*  ~ {LinkedWith:TIID^Device 3 (NOV/DP-RAM)^Outputs^Var 283} *)
	.SHADE3 AT %QB3112 : STRING(80);	(*  ~ {LinkedWith:TIID^Device 3 (NOV/DP-RAM)^Outputs^Var 289} *)
	.CONETIP3 AT %QB3196 : STRING(80);	(*  ~ {LinkedWith:TIID^Device 3 (NOV/DP-RAM)^Outputs^Var 295} *)
	.CONELENGTH3 AT %QB3280 : REAL;	(*  ~ {LinkedWith:TIID^Device 3 (NOV/DP-RAM)^Outputs^Var 327} *)
	.CONENETWT3 AT %QB3284 : REAL;	(*  ~ {LinkedWith:TIID^Device 3 (NOV/DP-RAM)^Outputs^Var 328} *)
	.DFLTNETWT3 AT %QB3288 : REAL;	(*  ~ {LinkedWith:TIID^Device 3 (NOV/DP-RAM)^Outputs^Var 344} *)
	.NETWTTOL3 AT %QB3292 : REAL;	(*  ~ {LinkedWith:TIID^Device 3 (NOV/DP-RAM)^Outputs^Var 345} *)
	.DFLTGROSSWT3 AT %QB3296 : REAL;	(*  ~ {LinkedWith:TIID^Device 3 (NOV/DP-RAM)^Outputs^Var 346} *)
	.GROSSWTTOL3 AT %QB3300 : REAL;	(*  ~ {LinkedWith:TIID^Device 3 (NOV/DP-RAM)^Outputs^Var 347} *)
	.NegTol3 AT %QB3304 : REAL;
	.PRGNO4 AT %QB3308 : DINT;	(*  ~ {LinkedWith:TIID^Device 3 (NOV/DP-RAM)^Outputs^Var 313} *)
	.COUNT4 AT %QB3312 : STRING(80);	(*  ~ {LinkedWith:TIID^Device 3 (NOV/DP-RAM)^Outputs^Var 265} *)
	.DETAILS4 AT %QB3396 : STRING(80);
	.LOTNO4 AT %QB3480 : STRING(80);	(*  ~ {LinkedWith:TIID^Device 3 (NOV/DP-RAM)^Outputs^Var 272} *)
	.CARTONNO4 AT %QB3564 : DINT;	(*  ~ {LinkedWith:TIID^Device 3 (NOV/DP-RAM)^Outputs^Var 319} *)
	.WORKORDERNO4 AT %QB3568 : STRING(80);	(*  ~ {LinkedWith:TIID^Device 3 (NOV/DP-RAM)^Outputs^Var 278} *)
	.BLEND4 AT %QB3652 : STRING(80);	(*  ~ {LinkedWith:TIID^Device 3 (NOV/DP-RAM)^Outputs^Var 284} *)
	.SHADE4 AT %QB3736 : STRING(80);	(*  ~ {LinkedWith:TIID^Device 3 (NOV/DP-RAM)^Outputs^Var 290} *)
	.CONETIP4 AT %QB3820 : STRING(80);	(*  ~ {LinkedWith:TIID^Device 3 (NOV/DP-RAM)^Outputs^Var 296} *)
	.CONELENGTH4 AT %QB3904 : REAL;	(*  ~ {LinkedWith:TIID^Device 3 (NOV/DP-RAM)^Outputs^Var 329} *)
	.DFLTNETWT4 AT %QB3908 : REAL;	(*  ~ {LinkedWith:TIID^Device 3 (NOV/DP-RAM)^Outputs^Var 348} *)
	.NETWTTOL4 AT %QB3912 : REAL;	(*  ~ {LinkedWith:TIID^Device 3 (NOV/DP-RAM)^Outputs^Var 349} *)
	.DFLTGROSSWT4 AT %QB3916 : REAL;	(*  ~ {LinkedWith:TIID^Device 3 (NOV/DP-RAM)^Outputs^Var 350} *)
	.GROSSWTTOL4 AT %QB3920 : REAL;	(*  ~ {LinkedWith:TIID^Device 3 (NOV/DP-RAM)^Outputs^Var 351} *)
	.NegTol4 AT %QB3924 : REAL;
	.PRGNO5 AT %QB3928 : DINT;	(*  ~ {LinkedWith:TIID^Device 3 (NOV/DP-RAM)^Outputs^Var 314} *)
	.COUNT5 AT %QB3932 : STRING(80);	(*  ~ {LinkedWith:TIID^Device 3 (NOV/DP-RAM)^Outputs^Var 266} *)
	.DETAILS5 AT %QB4016 : STRING(80);
	.LOTNO5 AT %QB4100 : STRING(80);	(*  ~ {LinkedWith:TIID^Device 3 (NOV/DP-RAM)^Outputs^Var 273} *)
	.CARTONNO5 AT %QB4184 : DINT;	(*  ~ {LinkedWith:TIID^Device 3 (NOV/DP-RAM)^Outputs^Var 320} *)
	.WORKORDERNO5 AT %QB4188 : STRING(80);	(*  ~ {LinkedWith:TIID^Device 3 (NOV/DP-RAM)^Outputs^Var 279} *)
	.BLEND5 AT %QB4272 : STRING(80);	(*  ~ {LinkedWith:TIID^Device 3 (NOV/DP-RAM)^Outputs^Var 285} *)
	.SHADE5 AT %QB4356 : STRING(80);	(*  ~ {LinkedWith:TIID^Device 3 (NOV/DP-RAM)^Outputs^Var 291} *)
	.CONETIP5 AT %QB4440 : STRING(80);	(*  ~ {LinkedWith:TIID^Device 3 (NOV/DP-RAM)^Outputs^Var 297} *)
	.CONELENGTH5 AT %QB4524 : REAL;	(*  ~ {LinkedWith:TIID^Device 3 (NOV/DP-RAM)^Outputs^Var 330} *)
	.CONENETWT5 AT %QB4528 : REAL;	(*  ~ {LinkedWith:TIID^Device 3 (NOV/DP-RAM)^Outputs^Var 331} *)
	.DFLTNETWT5 AT %QB4532 : REAL;	(*  ~ {LinkedWith:TIID^Device 3 (NOV/DP-RAM)^Outputs^Var 352} *)
	.NETWTTOL5 AT %QB4536 : REAL;	(*  ~ {LinkedWith:TIID^Device 3 (NOV/DP-RAM)^Outputs^Var 353} *)
	.DFLTGROSSWT5 AT %QB4540 : REAL;	(*  ~ {LinkedWith:TIID^Device 3 (NOV/DP-RAM)^Outputs^Var 354} *)
	.GROSSWTTOL5 AT %QB4544 : REAL;	(*  ~ {LinkedWith:TIID^Device 3 (NOV/DP-RAM)^Outputs^Var 355} *)
	.NegTol5 AT %QB4548 : REAL;
	.DOM_EXPORT AT %QB4552 : STRING(80);
	.PACKTYPE AT %QB4636 : STRING(80);
	.DOM_EXPORT1 AT %QB4720 : STRING(80);	(*  ~ {LinkedWith:TIID^Device 3 (NOV/DP-RAM)^Outputs^Var 299} *)
	.PACKTYPE1 AT %QB4804 : STRING(80);	(*  ~ {LinkedWith:TIID^Device 3 (NOV/DP-RAM)^Outputs^Var 305} *)
	.DOM_EXPORT2 AT %QB4888 : STRING(80);	(*  ~ {LinkedWith:TIID^Device 3 (NOV/DP-RAM)^Outputs^Var 300} *)
	.PACKTYPE2 AT %QB4972 : STRING(80);	(*  ~ {LinkedWith:TIID^Device 3 (NOV/DP-RAM)^Outputs^Var 306} *)
	.DOM_EXPORT3 AT %QB5056 : STRING(80);	(*  ~ {LinkedWith:TIID^Device 3 (NOV/DP-RAM)^Outputs^Var 301} *)
	.PACKTYPE3 AT %QB5140 : STRING(80);	(*  ~ {LinkedWith:TIID^Device 3 (NOV/DP-RAM)^Outputs^Var 307} *)
	.DOM_EXPORT4 AT %QB5224 : STRING(80);	(*  ~ {LinkedWith:TIID^Device 3 (NOV/DP-RAM)^Outputs^Var 302} *)
	.PACKTYPE4 AT %QB5308 : STRING(80);	(*  ~ {LinkedWith:TIID^Device 3 (NOV/DP-RAM)^Outputs^Var 308} *)
	.DOM_EXPORT5 AT %QB5392 : STRING(80);	(*  ~ {LinkedWith:TIID^Device 3 (NOV/DP-RAM)^Outputs^Var 303} *)
	.DOM_EXPORT_DIS AT %QB5476 : STRING(80);	(*  ~ {LinkedWith:TIID^Device 3 (NOV/DP-RAM)^Outputs^Var 298} *)
	.PACKTYPE5 AT %QB5560 : STRING(80);	(*  ~ {LinkedWith:TIID^Device 3 (NOV/DP-RAM)^Outputs^Var 309} *)
	.PACKTYPE_DIS AT %QB5644 : STRING(80);	(*  ~ {LinkedWith:TIID^Device 3 (NOV/DP-RAM)^Outputs^Var 304} *)
	.PRG1RUNNING AT %QX5749.5 : BOOL;	(*  ~ {LinkedWith:TIID^Device 3 (NOV/DP-RAM)^Outputs^Var 730} *)
	.PRG2RUNNING AT %QX5749.6 : BOOL;	(*  ~ {LinkedWith:TIID^Device 3 (NOV/DP-RAM)^Outputs^Var 731} *)
	.PRG3RUNNING AT %QX5749.7 : BOOL;	(*  ~ {LinkedWith:TIID^Device 3 (NOV/DP-RAM)^Outputs^Var 732} *)
	.PRG4RUNNING AT %QX5750.0 : BOOL;	(*  ~ {LinkedWith:TIID^Device 3 (NOV/DP-RAM)^Outputs^Var 733} *)
	.PRG5RUNNING AT %QX5750.1 : BOOL;	(*  ~ {LinkedWith:TIID^Device 3 (NOV/DP-RAM)^Outputs^Var 734} *)
	.SerialNo AT %QB5728 : DINT;
	.DefaultNetWt AT %QB5732 : REAL;
	.NetWtTolRep AT %QB5736 : REAL;
	.DefaultGrossWt AT %QB5740 : REAL;
	.GrossWtTolRep AT %QB5744 : REAL;
END_VAR

(* Data type *)
TYPE Production_Data :
STRUCT

	S_No						:STRING;
	ConeType					:STRING;
	CartonNo					:STRING;
	LotNo						:STRING;
	SDateF						:STRING;
	NetWt						:STRING;
	WorkOrderNo				:STRING;
	DefaultNettWeight				:STRING;
	DefaultGrossWeight			:STRING;
	Blend						:STRING;
	Shade						:STRING;
	ConeTip						:STRING;
	ConeNettWeight				:STRING;
	ConeLength					:STRING;
	Dom_Exp					:STRING;
	PackType					:STRING;
	CountCode					:STRING;


END_STRUCT
END_TYPE

(* Data type *)
TYPE ProductionData_IndoPrint1 :
STRUCT
	(*S_NO				:STRING;
	S_DATE				:STRING;
	CONETYPE			:STRING;
	CARTONNO			:STRING;
	LOTNO				:STRING;
	NETWT				:STRING;
	WORKORDERNO		:STRING;
	DFLTNTWT			:STRING;
	DFLTGRSWT		:STRING;
	BLEND				:STRING;
	SHADE 				:STRING;
	CONETIP 			:STRING;
	CONENTWT 			:STRING;
	CONELENGTH		 :STRING;
	DOMEXP 			:STRING;
	PACKTYPE 			:STRING;
	COUNTCODE 		:STRING;*)
	SERIALNO			:STRING;
	SDATE				:STRING;
	NOOFCONE				:STRING;
	BAGNO				:STRING;
	COUNTCODE		:STRING;
	LOTNO				:STRING;
	DFLTNETWEIGHT	:STRING;
	DFLTGRSST		:STRING;
	ACTWT	:STRING;
	BLND	:STRING;
	SHD		:STRING;
	CONTIP				:STRING;
	CONNETWT	:STRING;
	CONLEN		:STRING;
	DOM	:STRING;
	ITEMCODE:STRING;
	PACKTYP	:STRING;
	WRKORNO	:STRING;
	COUNT	:STRING;
	TAREWEIGHTDET:STRING;
	WORKFLAGDET	:STRING;
	ISSUEDESPATCH	:STRING;
	REMARKSDET:STRING;
	LOCATIONDET	:STRING;
	DESCRIPTION	:STRING;
	FINYEAR	:STRING;
	AVERAGEGCOUNT	:STRING;
	BARCODE:STRING;




END_STRUCT
END_TYPE

(* Data type *)
TYPE ProductionData_PrintData :
STRUCT
	(*Print:STRING;
	ConeType1:STRING;
	Blend1:STRING;
	DefaultnetWt1:STRING;
	DefaultGrossWt1:STRING;
	LotNo1:STRING;
	BagNo1:STRING;
	Shade1:STRING;
	ConeTip1:STRING;
	PackType1:STRING;
	Cones1:STRING;*)
	Print:STRING;
	PgNo:STRING;
	TotNoCones:STRING;
	CartNo:STRING;
	LotNo:STRING;
	DateTi:STRING;
	NetWt:STRING;
	WrkOrdNo:STRING;

	DfltNetWt:STRING;
	DfltGrsWt:STRING;
	Blnd:STRING;
	Shd:STRING;
	ConeTip:STRING;
	ConeNetWt:STRING;
	ConeLenght:STRING;
	Dom:STRING;
	Pack:STRING;
	CountCod:STRING;

END_STRUCT
END_TYPE

(* Data type *)
TYPE ProductionDataError_IndoPrint1 :
STRUCT
	SERIALNOERROR:STRING;
	SDATEERROR:STRING;
	STIMEEROOR:STRING;
	SHIFTERROR:STRING;
	ERRORIDERROR:STRING;
END_STRUCT
END_TYPE

(* Data type *)
TYPE ST_CSV_Record :
STRUCT
	sName 	: T_MaxString 	:= '';
	nNumber	: UDINT 		:= 0;
	fPos		: LREAL 		:= 0.0;
	bOP		: BOOL 		:= FALSE;
	sDesc		: STRING(40)	:= '';
	data		: ARRAY[0..7] OF STRING;
END_STRUCT
END_TYPE

(* POU MAIN, ST *)
PROGRAM MAIN
VAR
	bTestBool: BOOL;
END_VAR
(*================== Model Selection Logic==========*)
IF bIAutoManual THEN bAutoModeOn:=TRUE; sAMcModeStatus:='Machine In Auto Mode'; bManualModeOn:=FALSE;

ELSIF NOT bIAutoManual THEN bManualModeOn:=TRUE;  sAMcModeStatus:='Machine In Manual Mode'; bAutoModeOn:=FALSE; END_IF


DATALOG_REPORT();
DATAERRORLOG_REPORT();
Date_Time();
Parameters();
DATALOG_PRINT();
One_Min_Conv();
FlimRollerUnit();
Auto();
UnitA_RowStopper();
UnitB_RowStopper();
Manual();
Outputs();
ConeFeedPiston();
ConeFeedConv();
Serial();
FwdPiston();

Wrapping_Unit();
Sealing_Unit();
Sealing_Conveyor();
WeightCalc();

INT_All();
Cylinder_Alarm();
ConeAllignAlarm();
ConeMiss_Alarm();
Common();

DataLog_1();

(*-===========Sealing Complete delay from Hmi==================*)

SealComDlyTemp:= REAL_TO_TIME(rSealCompDlyHmi * 1000);


(*==========Pause & Reume Logic====================*)


	IF bPauseHmi  OR bAPauseEnable THEN bAPauseSeq:=TRUE; END_IF
	IF bResumeHmi THEN bAPauseSeq:=FALSE; END_IF
END_PROGRAM

(* POU AutoMode/DATALOG_REPORT, ST *)
PROGRAM DATALOG_REPORT
VAR
	R_TRIG_IndoPrint: R_TRIG;
	FB_FileOpen_Indo: FB_FileOpen;
	FB_FileWrite_Indo: FB_FileWrite;
	FB_FileClose_Indo: FB_FileClose;
	FB_FileDelete_Indo: FB_FileDelete;
	IndoReport: INT;
	ReportHead1_Indo: BOOL;
	ST1_ProductionData: BOOL;
	ReportHead2_Indo: BOOL;
	ReportBot1_Indo: BOOL;
	stStation1_ProductionData: BOOL;
	ReportBot2_Indo: BOOL;
	testbit: BOOL;
	TON_Indo1: TON;
	TON_Indo2: TON;
	TON_Indo3: TON;
	TON_Indo4: TON;
	sOldDay: STRING;
	TON_Newdaydly: TON;
	TON_NEWDAY: TON;

	TON_NewdaydlyError: TON;
	WriteError: INT;
	TON_writedly: TON;
	OpenError: INT;
	TON_Opendly: TON;

	BarcodeNo: STRING;
	BarCode1: STRING;
	EmptyConeWtRep: REAL;
	EmptyConeWtRep1: REAL;
END_VAR
FB_FileOpen_Indo(
	sNetId:='192.168.225.201.1.1',
	sPathName:= ReportPath_Final_2,
	nMode:=FOPEN_MODEAPPEND ,
	ePath:=PATH_GENERIC ,
	bExecute:= ,
	tTimeout:=T#2s ,
	bBusy=> ,
	bError=> ,
	nErrId=> ,
	hFile=> );

FB_FileWrite_Indo(
	sNetId:='	192.168.225.201.1.1',
	hFile:=FB_FileOpen_Indo.hFile ,
	pWriteBuff:=ADR(ProductionDataValues_IndoPrint_Com),
	cbWriteLen:=LEN(ProductionDataValues_IndoPrint_Com),
	bExecute:= ,
	tTimeout:=T#2s ,
	bBusy=> ,
	bError=> ,
	nErrId=> ,
	cbWrite=> );


FB_FileClose_Indo(
	sNetId:='192.168.225.201.1.1',
	hFile:=FB_FileOpen_Indo.hFile ,
	bExecute:= ,
	tTimeout:=T#2s ,
	bBusy=> ,
	bError=> ,
	nErrId=> );

FB_FileDelete_Indo(
	sNetId:='192.168.225.201.1.1' ,
	sPathName:= ReportPath_Final_2,
	ePath:=PATH_GENERIC ,
	bExecute:= ,
	tTimeout:=T#2s ,
	bBusy=> ,
	bError=> ,
	nErrId=> );

R_TRIG_IndoPrint(CLK:=( bANewDay OR testbit)  , Q=> );


CASE IndoReport OF
0:	  IF TON_NEWDAY.Q   THEN	sOldDay := sDay;TON_Newdaydly(IN:=TRUE , PT:=t#0.2s , Q=> , ET=> );
		IF TON_Newdaydly.Q THEN
		bANewDay:=FALSE;IndoReport:=1; SerialNoError:=1;FB_FileOpen_Indo.bExecute:=TRUE;END_IF END_IF

1:	TON_Newdaydly(IN:=FALSE);TON_NEWDAY(IN:=FALSE);
	IF NOT FB_FileOpen_Indo.bBusy AND NOT FB_FileOpen_Indo.bError AND FB_FileOpen_Indo.hFile>0 THEN ReportHead1_Indo:=TRUE;END_IF

	IF ReportHead1_Indo THEN
	ProductionData_IndoPrint:= CONCAT( 'DATE',',');
	ProductionData_IndoPrint:=	 CONCAT( ProductionData_IndoPrint,'DOM ');
		ProductionData_IndoPrint:= CONCAT( ProductionData_IndoPrint,',');
	ProductionData_IndoPrint:=	 CONCAT( ProductionData_IndoPrint,'BAG NO');
		ProductionData_IndoPrint:= CONCAT( ProductionData_IndoPrint,',');
	ProductionData_IndoPrint:=	 CONCAT( ProductionData_IndoPrint,' PACK');
		ProductionData_IndoPrint:= CONCAT( ProductionData_IndoPrint,',');
	ProductionData_IndoPrint:=	 CONCAT( ProductionData_IndoPrint,'ITEM CODE');
		ProductionData_IndoPrint:=CONCAT( ProductionData_IndoPrint,',');
	ProductionData_IndoPrint:=	 CONCAT( ProductionData_IndoPrint,'LOT NO');
		ProductionData_IndoPrint:=CONCAT( ProductionData_IndoPrint,',');
	ProductionData_IndoPrint:=	 CONCAT( ProductionData_IndoPrint,'COUNT');
		ProductionData_IndoPrint:=CONCAT( ProductionData_IndoPrint,',');

ProductionData_IndoPrint:=	 CONCAT( ProductionData_IndoPrint,'BLEND');
		ProductionData_IndoPrint:=CONCAT( ProductionData_IndoPrint,',');

ProductionData_IndoPrint:=	 CONCAT( ProductionData_IndoPrint,'SHDAE');
		ProductionData_IndoPrint:=CONCAT( ProductionData_IndoPrint,',');


ProductionData_IndoPrint:=	 CONCAT( ProductionData_IndoPrint,'CONES');
		ProductionData_IndoPrint:=CONCAT( ProductionData_IndoPrint,',');

ProductionData_IndoPrint:=	 CONCAT( ProductionData_IndoPrint,'NET WT');
		ProductionData_IndoPrint:=CONCAT( ProductionData_IndoPrint,',');

ProductionData_IndoPrint:=	 CONCAT( ProductionData_IndoPrint,'TARE WT');
		ProductionData_IndoPrint:=CONCAT( ProductionData_IndoPrint,',');


ProductionData_IndoPrint:=	 CONCAT( ProductionData_IndoPrint,'GR WT');
		ProductionData_IndoPrint:=CONCAT( ProductionData_IndoPrint,',');


ProductionData_IndoPrint:=	 CONCAT( ProductionData_IndoPrint,'CN WT');
		ProductionData_IndoPrint:=CONCAT( ProductionData_IndoPrint,',');

ProductionData_IndoPrint:=	 CONCAT( ProductionData_IndoPrint,'CN LEN');
		ProductionData_IndoPrint:=CONCAT( ProductionData_IndoPrint,',');

ProductionData_IndoPrint:=	 CONCAT( ProductionData_IndoPrint,'WORK ORDER');
		ProductionData_IndoPrint:=CONCAT( ProductionData_IndoPrint,',');

ProductionData_IndoPrint:=	 CONCAT( ProductionData_IndoPrint,'BAR CODE');
		ProductionData_IndoPrint:=CONCAT( ProductionData_IndoPrint,',');

	ProductionData_IndoPrint:=	 CONCAT( ProductionData_IndoPrint,'WORCP FLAG');
ProductionData_IndoPrint:=CONCAT( ProductionData_IndoPrint,',');
		(*ProductionData_IndoPrint:= CONCAT( ProductionData_IndoPrint,'$0A');*)
(*ProductionData_IndoPrint:=	 CONCAT( ProductionData_IndoPrint,'DFLT GROSS WT');
		ProductionData_IndoPrint:=CONCAT( ProductionData_IndoPrint,',');
ProductionData_IndoPrint:=	 CONCAT( ProductionData_IndoPrint,'ACT GROSS WT');
		ProductionData_IndoPrint:= CONCAT( ProductionData_IndoPrint,'$0A');
ProductionData_IndoPrint:=	 CONCAT( ProductionData_IndoPrint,'Cn9Wt');
		ProductionData_IndoPrint:=CONCAT( ProductionData_IndoPrint,',');
ProductionData_IndoPrint:=	 CONCAT( ProductionData_IndoPrint,'Cn10Wt');
		ProductionData_IndoPrint:=CONCAT( ProductionData_IndoPrint,',');
ProductionData_IndoPrint:=	 CONCAT( ProductionData_IndoPrint,'Cn11Wt');
		ProductionData_IndoPrint:=CONCAT( ProductionData_IndoPrint,',');
ProductionData_IndoPrint:=	 CONCAT( ProductionData_IndoPrint,'Cn12Wt');
	ProductionData_IndoPrint:=CONCAT( ProductionData_IndoPrint,',');*)
IndoReport:=2; END_IF

2:	PROCESSCOMPLETE:=FALSE;ReportHead1_Indo:=FALSE;ProductionDataValues_IndoPrint_Com:=ProductionData_IndoPrint;
	TON_Indo1(IN:=TRUE , PT:=t#5s , Q=> , ET=> );
	FB_FileWrite_Indo.bExecute:=TRUE;
	IF NOT FB_FileWrite_Indo.bBusy AND NOT FB_FileWrite_Indo.bError AND FB_FileWrite_Indo.hFile>0 AND TON_Indo1.Q THEN IndoReport:=IndoReport+1; END_IF

3:	ProductionDataValues_IndoPrint_Com:=ProductionData_IndoPrint;
	FB_FileWrite_Indo.bExecute:=TRUE;
	IF NOT FB_FileWrite_Indo.bBusy AND NOT FB_FileWrite_Indo.bError THEN IndoReport:=IndoReport+1; END_IF

4:	FB_FileWrite_Indo.bExecute:=FALSE;ProductionData_IndoPrint:='';IndoReport:=IndoReport+1;

5:	ReportHead2_Indo:=TRUE;
	IF ReportHead2_Indo THEN IndoReport:=IndoReport+1;END_IF

6:	ProductionData_IndoPrint:=	 CONCAT( ProductionData_IndoPrint,'ISSUE DESP');
		ProductionData_IndoPrint:=CONCAT( ProductionData_IndoPrint,',');
ProductionData_IndoPrint:=	 CONCAT( ProductionData_IndoPrint,'LOCATION');
		ProductionData_IndoPrint:=CONCAT( ProductionData_IndoPrint,',');
ProductionData_IndoPrint:=	 CONCAT( ProductionData_IndoPrint,'REMARKS');
		ProductionData_IndoPrint:=CONCAT( ProductionData_IndoPrint,',');
ProductionData_IndoPrint:=	 CONCAT( ProductionData_IndoPrint,'ITEM DESCR');
		ProductionData_IndoPrint:=CONCAT( ProductionData_IndoPrint,',');
ProductionData_IndoPrint:=	 CONCAT( ProductionData_IndoPrint,'CN TIP');
		ProductionData_IndoPrint:=CONCAT( ProductionData_IndoPrint,',');
ProductionData_IndoPrint:=	 CONCAT( ProductionData_IndoPrint,'ACT WT');
		ProductionData_IndoPrint:=CONCAT( ProductionData_IndoPrint,',');
ProductionData_IndoPrint:=	 CONCAT( ProductionData_IndoPrint,'FYEAR');
		ProductionData_IndoPrint:=CONCAT( ProductionData_IndoPrint,',');
(*ProductionData_IndoPrint:=	 CONCAT( ProductionData_IndoPrint,'Cn20Wt');
		ProductionData_IndoPrint:=CONCAT( ProductionData_IndoPrint,',');
ProductionData_IndoPrint:=	 CONCAT( ProductionData_IndoPrint,'Cn21Wt');
		ProductionData_IndoPrint:=CONCAT( ProductionData_IndoPrint,',');
ProductionData_IndoPrint:=	 CONCAT( ProductionData_IndoPrint,'Cn22Wt');
		ProductionData_IndoPrint:=CONCAT( ProductionData_IndoPrint,',');
ProductionData_IndoPrint:=	 CONCAT( ProductionData_IndoPrint,'Cn23Wt');
		ProductionData_IndoPrint:=CONCAT( ProductionData_IndoPrint,',');*)
	ProductionData_IndoPrint:=	 CONCAT( ProductionData_IndoPrint,'AVG COUNT');
ProductionData_IndoPrint:= CONCAT( ProductionData_IndoPrint,'$0A');
ReportHead2_Indo:=FALSE;
IndoReport:=IndoReport+1;

7:	ReportHead1_Indo:=FALSE;ProductionDataValues_IndoPrint_Com:=ProductionData_IndoPrint;
TON_Indo2(IN:=TRUE , PT:=t#5s , Q=> , ET=> );
	FB_FileWrite_Indo.bExecute:=TRUE;
	IF NOT FB_FileWrite_Indo.bBusy AND NOT FB_FileWrite_Indo.bError  AND TON_Indo2.Q THEN  IndoReport:=IndoReport+1; END_IF

8:	FB_FileWrite_Indo.bExecute:=FALSE;
	FB_FileClose_Indo.bExecute:=TRUE;
	 IF NOT FB_FileClose_Indo.bBusy AND NOT FB_FileClose_Indo.bError THEN FB_FileOpen_Indo.bExecute:=FALSE; IndoReport:=IndoReport+1;END_IF(*ProductionData_IndoPrint:='';*)

9:	FB_FileClose_Indo.bExecute:=FALSE;
	IF ReportSave OR testbit THEN

	FB_FileOpen_Indo.bExecute:=TRUE;
	IF NOT FB_FileOpen_Indo.bBusy AND NOT FB_FileOpen_Indo.bError AND FB_FileOpen_Indo.hFile>0 THEN  ReportBot1_Indo:=TRUE;END_IF

	IF ReportBot1_Indo THEN IndoReport:=IndoReport+1;END_IF END_IF

10:
ProductionData_IndoPrint2:= CONCAT(ProductionData_IndoPrint11.SDATE,',');
ProductionData_IndoPrint2:=	 CONCAT( ProductionData_IndoPrint2,ProductionData_IndoPrint11.DOM);
ProductionData_IndoPrint2:= CONCAT( ProductionData_IndoPrint2,',');
ProductionData_IndoPrint2:=	 CONCAT( ProductionData_IndoPrint2,ProductionData_IndoPrint11.BAGNO	);
ProductionData_IndoPrint2:= CONCAT( ProductionData_IndoPrint2,',');
ProductionData_IndoPrint2:=	 CONCAT( ProductionData_IndoPrint2,ProductionData_IndoPrint11.PACKTYP	);
ProductionData_IndoPrint2:= CONCAT( ProductionData_IndoPrint2,',');
ProductionData_IndoPrint2:=	 CONCAT( ProductionData_IndoPrint2,ProductionData_IndoPrint11.ITEMCODE);
ProductionData_IndoPrint2:= CONCAT( ProductionData_IndoPrint2,',');
ProductionData_IndoPrint2:=	 CONCAT( ProductionData_IndoPrint2,ProductionData_IndoPrint11.LOTNO);
ProductionData_IndoPrint2:= CONCAT( ProductionData_IndoPrint2,',');
ProductionData_IndoPrint2:=	 CONCAT( ProductionData_IndoPrint2,ProductionData_IndoPrint11.COUNT);
ProductionData_IndoPrint2:= CONCAT( ProductionData_IndoPrint2,',');

ProductionData_IndoPrint2:=	 CONCAT( ProductionData_IndoPrint2,ProductionData_IndoPrint11.BLND);
ProductionData_IndoPrint2:= CONCAT( ProductionData_IndoPrint2,',');

ProductionData_IndoPrint2:=	 CONCAT( ProductionData_IndoPrint2,ProductionData_IndoPrint11.SHD);
ProductionData_IndoPrint2:= CONCAT( ProductionData_IndoPrint2,',');
(*

ProductionData_IndoPrint2:=	 CONCAT( ProductionData_IndoPrint2,ProductionData_IndoPrint11.BLND);
ProductionData_IndoPrint2:= CONCAT( ProductionData_IndoPrint2,',');


ProductionData_IndoPrint2:=	 CONCAT( ProductionData_IndoPrint2,ProductionData_IndoPrint11.SHD);
ProductionData_IndoPrint2:= CONCAT( ProductionData_IndoPrint2,',');
*)

ProductionData_IndoPrint2:=	 CONCAT( ProductionData_IndoPrint2,ProductionData_IndoPrint11.NOOFCONE);
ProductionData_IndoPrint2:= CONCAT( ProductionData_IndoPrint2,',');


ProductionData_IndoPrint2:=	 CONCAT( ProductionData_IndoPrint2,ProductionData_IndoPrint11.DFLTNETWEIGHT);
ProductionData_IndoPrint2:= CONCAT( ProductionData_IndoPrint2,',');


ProductionData_IndoPrint2:=	 CONCAT( ProductionData_IndoPrint2,ProductionData_IndoPrint11.TAREWEIGHTDET);
ProductionData_IndoPrint2:= CONCAT( ProductionData_IndoPrint2,',');


ProductionData_IndoPrint2:=	 CONCAT( ProductionData_IndoPrint2,ProductionData_IndoPrint11.DFLTGRSST);
ProductionData_IndoPrint2:= CONCAT( ProductionData_IndoPrint2,',');


ProductionData_IndoPrint2:=	 CONCAT( ProductionData_IndoPrint2,ProductionData_IndoPrint11.CONNETWT);
ProductionData_IndoPrint2:= CONCAT( ProductionData_IndoPrint2,',');


ProductionData_IndoPrint2:=	 CONCAT( ProductionData_IndoPrint2,ProductionData_IndoPrint11.CONLEN);
ProductionData_IndoPrint2:= CONCAT( ProductionData_IndoPrint2,',');


ProductionData_IndoPrint2:=	 CONCAT( ProductionData_IndoPrint2,ProductionData_IndoPrint11.WRKORNO);
ProductionData_IndoPrint2:= CONCAT( ProductionData_IndoPrint2,',');
(*ProductionData_IndoPrint2:= CONCAT( ProductionData_IndoPrint2,'$0A');*)

ReportBot1_Indo:=FALSE;ReportSave:=FALSE;
IndoReport:=11;


11:	ProductionDataValues_IndoPrint_Com:=ProductionData_IndoPrint2;
	TON_Indo3(IN:=TRUE , PT:=t#5s , Q=> , ET=> );
	FB_FileWrite_Indo.bExecute:=TRUE;
	IF NOT FB_FileWrite_Indo.bBusy AND NOT FB_FileWrite_Indo.bError AND TON_Indo3.Q THEN IndoReport:=IndoReport+1; END_IF

12:	FB_FileWrite_Indo.bExecute:=FALSE;(*ProductionData_IndoPrint:='';*)IndoReport:=IndoReport+1;

13:	ReportBot2_Indo:=TRUE;
	IF ReportBot2_Indo THEN IndoReport:=IndoReport+1;END_IF

14:ProductionData_IndoPrint2:= CONCAT(ProductionData_IndoPrint11.BARCODE,',');
ProductionData_IndoPrint2:=	 CONCAT( ProductionData_IndoPrint2,ProductionData_IndoPrint11.WORKFLAGDET);
ProductionData_IndoPrint2:= CONCAT( ProductionData_IndoPrint2,',');
ProductionData_IndoPrint2:=	 CONCAT( ProductionData_IndoPrint2,ProductionData_IndoPrint11.ISSUEDESPATCH);
ProductionData_IndoPrint2:= CONCAT( ProductionData_IndoPrint2,',');
ProductionData_IndoPrint2:=	 CONCAT( ProductionData_IndoPrint2,ProductionData_IndoPrint11.LOCATIONDET);
ProductionData_IndoPrint2:= CONCAT( ProductionData_IndoPrint2,',');
ProductionData_IndoPrint2:=	 CONCAT( ProductionData_IndoPrint2,ProductionData_IndoPrint11.REMARKSDET);
ProductionData_IndoPrint2:= CONCAT( ProductionData_IndoPrint2,',');
ProductionData_IndoPrint2:=	 CONCAT( ProductionData_IndoPrint2,ProductionData_IndoPrint11.DESCRIPTION);
ProductionData_IndoPrint2:= CONCAT( ProductionData_IndoPrint2,',');
ProductionData_IndoPrint2:=	 CONCAT( ProductionData_IndoPrint2,ProductionData_IndoPrint11.CONTIP);
ProductionData_IndoPrint2:= CONCAT( ProductionData_IndoPrint2,',');
ProductionData_IndoPrint2:=	 CONCAT( ProductionData_IndoPrint2,ProductionData_IndoPrint11.ACTWT);
ProductionData_IndoPrint2:= CONCAT( ProductionData_IndoPrint2,',');
ProductionData_IndoPrint2:=	 CONCAT( ProductionData_IndoPrint2,ProductionData_IndoPrint11.FINYEAR);
ProductionData_IndoPrint2:= CONCAT( ProductionData_IndoPrint2,',');
(*ProductionData_IndoPrint2:=	 CONCAT( ProductionData_IndoPrint2,ProductionData_IndoPrint11.NetWt21);
ProductionData_IndoPrint2:= CONCAT( ProductionData_IndoPrint2,',');
ProductionData_IndoPrint2:=	 CONCAT( ProductionData_IndoPrint2,ProductionData_IndoPrint11.NetWt22);
ProductionData_IndoPrint2:= CONCAT( ProductionData_IndoPrint2,',');
ProductionData_IndoPrint2:=	 CONCAT( ProductionData_IndoPrint2,ProductionData_IndoPrint11.NetWt23);
ProductionData_IndoPrint2:= CONCAT( ProductionData_IndoPrint2,',');*)
ProductionData_IndoPrint2:=	 CONCAT( ProductionData_IndoPrint2,ProductionData_IndoPrint11.AVERAGEGCOUNT);
(*ProductionData_IndoPrint2:= CONCAT( ProductionData_IndoPrint2,',');*)
ProductionData_IndoPrint2:= CONCAT( ProductionData_IndoPrint2,'$0A');
ReportBot2_Indo:=FALSE;
IndoReport:=IndoReport+1;

15:ProductionDataValues_IndoPrint_Com:=ProductionData_IndoPrint2;
TON_Indo4(IN:=TRUE , PT:=t#5s , Q=> , ET=> );

	FB_FileWrite_Indo.bExecute:=TRUE; IndoReport:=IndoReport+1;
	(*IF NOT FB_FileWrite_Indo.bBusy AND NOT FB_FileWrite_Indo.bError AND TON_Indo4.Q  THEN IndoReport:=IndoReport+1;END_IF*)

16:	IF NOT FB_FileWrite_Indo.bBusy AND NOT FB_FileWrite_Indo.bError THEN FB_FileWrite_Indo.bExecute:=FALSE; IndoReport:=IndoReport+1;END_IF


17:	TON_Indo3(IN:=FALSE);TON_Indo4(IN:=FALSE);TON_Indo2(IN:=FALSE);TON_Indo1(IN:=FALSE);FB_FileWrite_Indo.bExecute:=FALSE;IndoReport:=IndoReport+1;

18:	FB_FileClose_Indo.bExecute:=TRUE;
	 IF NOT FB_FileClose_Indo.bBusy AND NOT FB_FileClose_Indo.bError THEN  IndoReport:=20;END_IF

19:	IF bANewDay THEN IndoReport:=IndoReport+1;
	ELSIF NOT bANewDay THEN FB_FileOpen_Indo.bExecute:=FALSE; IndoReport:=9;
END_IF

20:	FB_FileOpen_Indo.bExecute:=FALSE;SerialNo:=SerialNo+1;IndoReport:=9;

END_CASE



IF sDay <> sOldDay THEN bANewDay:=TRUE;IndoReport:=0; SerialNo:=0;END_IF
TON_NEWDAY(IN:=bANewDay , PT:=T#0.5s , Q=> , ET=> );




CASE WriteError OF

0:	IF FB_FileWrite_Indo.bError THEN FB_FileWrite_Indo.bExecute:=FALSE;TON_writedly(IN:=FALSE);
	WriteError:=WriteError+1;END_IF

1:	TON_writedly(IN:=TRUE , PT:=t#2s , Q=> , ET=> );
	IF TON_writedly.Q THEN FB_FileWrite_Indo.bExecute:=TRUE;WriteError:=WriteError+1;END_IF

2:	TON_writedly(IN:=FALSE);WriteError:=0;

END_CASE




CASE OpenError OF

0:	IF FB_FileOpen_Indo.bError THEN FB_FileOpen_Indo.bExecute:=FALSE;TON_Opendly(IN:=FALSE);
	OpenError:=OpenError+1;END_IF

1:	TON_Opendly(IN:=TRUE , PT:=t#2s , Q=> , ET=> );
	IF TON_Opendly.Q THEN FB_FileOpen_Indo.bExecute:=TRUE;OpenError:=OpenError+1;END_IF

2:	TON_Opendly(IN:=FALSE);OpenError:=0;

END_CASE

EmptyConeWtRep1:=(iATotalNoOfCones * EmptyConeWt_DIS);
EmptyConeWtRep:=(var_5  - EmptyConeWtRep1);

TareWeight:=(DFLTGROSSWT_DIS - DFLTNETWT_DIS);


BarCode1:=CONCAT(STR1:=LOTNO_DIS, STR2:='.');
BarCode:=CONCAT(STR1:=BarCode1, STR2:=(sBagNoRep));








	ProductionData_IndoPrint11.DOM	:= (DOM_EXPORT_DIS);
	ProductionData_IndoPrint11.BAGNO	:=DINT_TO_STRING(CARTONNO_DIS)(*CartonNoHmi*);
	ProductionData_IndoPrint11.PACKTYP	:=(PACKTYPE_DIS);
	ProductionData_IndoPrint11.ITEMCODE	:=(ItemCodeHmi_DIS);
	ProductionData_IndoPrint11.LOTNO	:=(LOTNO_DIS);
	ProductionData_IndoPrint11.COUNT	:=(COUNT_DIS);
	ProductionData_IndoPrint11.BLND	:=(BLEND_DIS);
	ProductionData_IndoPrint11.SHD	:=(SHADE_DIS );
	ProductionData_IndoPrint11.NOOFCONE	:=INT_TO_STRING( iATotalNoOfCones );
	ProductionData_IndoPrint11.DFLTNETWEIGHT	:=REAL_TO_STRING(DFLTNETWT_DIS);
	ProductionData_IndoPrint11.TAREWEIGHTDET	:=REAL_TO_STRING(TareWeight_DIS);
	ProductionData_IndoPrint11.DFLTGRSST	:=REAL_TO_STRING(DFLTGROSSWT_DIS);
	ProductionData_IndoPrint11.CONNETWT	:=REAL_TO_STRING(CONENETWT_DIS);
	ProductionData_IndoPrint11.CONLEN	:=REAL_TO_STRING (CONELENGTH_DIS);
	ProductionData_IndoPrint11.WRKORNO	:=(WORKORDERNO_DIS);
	ProductionData_IndoPrint11.BARCODE	:=(BarCode);
	ProductionData_IndoPrint11.WORKFLAGDET	:=(WorkFlag_DIS);
	ProductionData_IndoPrint11.ISSUEDESPATCH	:=(IssueDesp_DIS);
	ProductionData_IndoPrint11.LOCATIONDET	:=(Location_DIS);
	ProductionData_IndoPrint11.REMARKSDET	:=(Remarks_DIS);
	ProductionData_IndoPrint11.DESCRIPTION	:=(Description_DIS);
	ProductionData_IndoPrint11.CONTIP	:=(CONETIP_DIS);
	ProductionData_IndoPrint11.ACTWT	:=REAL_TO_STRING(EmptyConeWtRep);
	ProductionData_IndoPrint11.FINYEAR	:=(Fyear_DIS);
	ProductionData_IndoPrint11.AVERAGEGCOUNT	:=(AvgCount_DIS);

		ProductionData_IndoPrint11.SERIALNO	:=INT_TO_STRING(Pgm_NoHmi);
		ProductionData_IndoPrint11.SDATE	:=(sDaateReport);



(*
CASE IndoReport OF
0:	  IF TON_NEWDAY.Q   THEN	sOldDay := sDay;TON_Newdaydly(IN:=TRUE , PT:=t#0.2s , Q=> , ET=> );
		IF TON_Newdaydly.Q THEN
		bANewDay:=FALSE;IndoReport:=1; SerialNo:=1;BagSerialNo:=0;FB_FileOpen_Indo.bExecute:=TRUE;END_IF END_IF

1:	TON_Newdaydly(IN:=FALSE);TON_NEWDAY(IN:=FALSE);
	IF NOT FB_FileOpen_Indo.bBusy AND NOT FB_FileOpen_Indo.bError AND FB_FileOpen_Indo.hFile>0 THEN ReportHead1_Indo:=TRUE;END_IF

	IF ReportHead1_Indo THEN
	ProductionData_IndoPrint:= CONCAT( 'SL NO',',');
	ProductionData_IndoPrint:=	 CONCAT( ProductionData_IndoPrint,'DATE');
		ProductionData_IndoPrint:= CONCAT( ProductionData_IndoPrint,',');
	(*ProductionData_IndoPrint:=	 CONCAT( ProductionData_IndoPrint,'TIME');
		ProductionData_IndoPrint:=CONCAT( ProductionData_IndoPrint,',');*)
	ProductionData_IndoPrint:=	 CONCAT( ProductionData_IndoPrint,'NO OF CONES');
		ProductionData_IndoPrint:= CONCAT( ProductionData_IndoPrint,',');
	ProductionData_IndoPrint:=	 CONCAT( ProductionData_IndoPrint,'CARTON NO');
		ProductionData_IndoPrint:=CONCAT( ProductionData_IndoPrint,',');
	ProductionData_IndoPrint:=	 CONCAT( ProductionData_IndoPrint,'LOT NO');
		ProductionData_IndoPrint:=CONCAT( ProductionData_IndoPrint,',');
	ProductionData_IndoPrint:=	 CONCAT( ProductionData_IndoPrint,'NET WT');
		ProductionData_IndoPrint:=CONCAT( ProductionData_IndoPrint,',');
	ProductionData_IndoPrint:=	 CONCAT( ProductionData_IndoPrint,'WRK ORD NO');
		ProductionData_IndoPrint:=CONCAT( ProductionData_IndoPrint,',');
	ProductionData_IndoPrint:=	 CONCAT( ProductionData_IndoPrint,'DFLT NT WT');
		ProductionData_IndoPrint:=CONCAT( ProductionData_IndoPrint,',');
	ProductionData_IndoPrint:=	 CONCAT( ProductionData_IndoPrint,'DFLT GRS WT');
		ProductionData_IndoPrint:=CONCAT( ProductionData_IndoPrint,',');
	ProductionData_IndoPrint:=	 CONCAT( ProductionData_IndoPrint,'BLEND');
		ProductionData_IndoPrint:=CONCAT( ProductionData_IndoPrint,',');
	ProductionData_IndoPrint:=	 CONCAT( ProductionData_IndoPrint,'SHADE');
		ProductionData_IndoPrint:=CONCAT( ProductionData_IndoPrint,',');
	ProductionData_IndoPrint:=	 CONCAT( ProductionData_IndoPrint,'CONE TIP');
		ProductionData_IndoPrint:=CONCAT( ProductionData_IndoPrint,',');
	ProductionData_IndoPrint:=	 CONCAT( ProductionData_IndoPrint,'CONE NT WT');
		ProductionData_IndoPrint:=CONCAT( ProductionData_IndoPrint,',');
	ProductionData_IndoPrint:=	 CONCAT( ProductionData_IndoPrint,'CONE LENGTH');
		ProductionData_IndoPrint:=CONCAT( ProductionData_IndoPrint,',');
	ProductionData_IndoPrint:=	 CONCAT( ProductionData_IndoPrint,'DOM EXP');
		ProductionData_IndoPrint:=CONCAT( ProductionData_IndoPrint,',');
	ProductionData_IndoPrint:=	 CONCAT( ProductionData_IndoPrint,'PACK TYPE');
		ProductionData_IndoPrint:=CONCAT( ProductionData_IndoPrint,',');
	ProductionData_IndoPrint:=	 CONCAT( ProductionData_IndoPrint,'COUNT CODE');
		ProductionData_IndoPrint:= CONCAT( ProductionData_IndoPrint,'$0A');
(*ProductionData_IndoPrint:=	 CONCAT( ProductionData_IndoPrint,'DFLT GROSS WT');
		ProductionData_IndoPrint:=CONCAT( ProductionData_IndoPrint,',');
ProductionData_IndoPrint:=	 CONCAT( ProductionData_IndoPrint,'ACT GROSS WT');
		ProductionData_IndoPrint:= CONCAT( ProductionData_IndoPrint,'$0A');
ProductionData_IndoPrint:=	 CONCAT( ProductionData_IndoPrint,'Cn9Wt');
		ProductionData_IndoPrint:=CONCAT( ProductionData_IndoPrint,',');
ProductionData_IndoPrint:=	 CONCAT( ProductionData_IndoPrint,'Cn10Wt');
		ProductionData_IndoPrint:=CONCAT( ProductionData_IndoPrint,',');
ProductionData_IndoPrint:=	 CONCAT( ProductionData_IndoPrint,'Cn11Wt');
		ProductionData_IndoPrint:=CONCAT( ProductionData_IndoPrint,',');
ProductionData_IndoPrint:=	 CONCAT( ProductionData_IndoPrint,'Cn12Wt');
	ProductionData_IndoPrint:=CONCAT( ProductionData_IndoPrint,',');*)
IndoReport:=7; END_IF

2:	PROCESSCOMPLETE:=FALSE;ReportHead1_Indo:=FALSE;ProductionDataValues_IndoPrint_Com:=ProductionData_IndoPrint;
	TON_Indo1(IN:=TRUE , PT:=t#5s , Q=> , ET=> );
	FB_FileWrite_Indo.bExecute:=TRUE;
	IF NOT FB_FileWrite_Indo.bBusy AND NOT FB_FileWrite_Indo.bError AND FB_FileWrite_Indo.hFile>0 AND TON_Indo1.Q THEN IndoReport:=IndoReport+1; END_IF

3:	ProductionDataValues_IndoPrint_Com:=ProductionData_IndoPrint;
	FB_FileWrite_Indo.bExecute:=TRUE;
	IF NOT FB_FileWrite_Indo.bBusy AND NOT FB_FileWrite_Indo.bError THEN IndoReport:=IndoReport+1; END_IF

4:	FB_FileWrite_Indo.bExecute:=FALSE;ProductionData_IndoPrint:='';IndoReport:=IndoReport+1;

5:	ReportHead2_Indo:=TRUE;
	IF ReportHead2_Indo THEN IndoReport:=IndoReport+1;END_IF

6:	ProductionData_IndoPrint:=	 CONCAT( ProductionData_IndoPrint,'Cn13Wt');
		ProductionData_IndoPrint:=CONCAT( ProductionData_IndoPrint,',');
ProductionData_IndoPrint:=	 CONCAT( ProductionData_IndoPrint,'Cn14Wt');
		ProductionData_IndoPrint:=CONCAT( ProductionData_IndoPrint,',');
ProductionData_IndoPrint:=	 CONCAT( ProductionData_IndoPrint,'Cn15Wt');
		ProductionData_IndoPrint:=CONCAT( ProductionData_IndoPrint,',');
ProductionData_IndoPrint:=	 CONCAT( ProductionData_IndoPrint,'Cn16Wt');
		ProductionData_IndoPrint:=CONCAT( ProductionData_IndoPrint,',');
ProductionData_IndoPrint:=	 CONCAT( ProductionData_IndoPrint,'Cn17Wt');
		ProductionData_IndoPrint:=CONCAT( ProductionData_IndoPrint,',');
ProductionData_IndoPrint:=	 CONCAT( ProductionData_IndoPrint,'Cn18Wt');
		ProductionData_IndoPrint:=CONCAT( ProductionData_IndoPrint,',');
ProductionData_IndoPrint:=	 CONCAT( ProductionData_IndoPrint,'Cn19Wt');
		ProductionData_IndoPrint:=CONCAT( ProductionData_IndoPrint,',');
ProductionData_IndoPrint:=	 CONCAT( ProductionData_IndoPrint,'Cn20Wt');
		ProductionData_IndoPrint:=CONCAT( ProductionData_IndoPrint,',');
ProductionData_IndoPrint:=	 CONCAT( ProductionData_IndoPrint,'Cn21Wt');
		ProductionData_IndoPrint:=CONCAT( ProductionData_IndoPrint,',');
ProductionData_IndoPrint:=	 CONCAT( ProductionData_IndoPrint,'Cn22Wt');
		ProductionData_IndoPrint:=CONCAT( ProductionData_IndoPrint,',');
ProductionData_IndoPrint:=	 CONCAT( ProductionData_IndoPrint,'Cn23Wt');
		ProductionData_IndoPrint:=CONCAT( ProductionData_IndoPrint,',');
	ProductionData_IndoPrint:=	 CONCAT( ProductionData_IndoPrint,'Cn24Wt');
ProductionData_IndoPrint:= CONCAT( ProductionData_IndoPrint,'$0A');
ReportHead2_Indo:=FALSE;
IndoReport:=IndoReport+1;

7:	ReportHead1_Indo:=FALSE;ProductionDataValues_IndoPrint_Com:=ProductionData_IndoPrint;
TON_Indo2(IN:=TRUE , PT:=t#5s , Q=> , ET=> );
	FB_FileWrite_Indo.bExecute:=TRUE;
	IF NOT FB_FileWrite_Indo.bBusy AND NOT FB_FileWrite_Indo.bError  AND TON_Indo2.Q THEN  IndoReport:=IndoReport+1; END_IF

8:	FB_FileWrite_Indo.bExecute:=FALSE;
	FB_FileClose_Indo.bExecute:=TRUE;
	 IF NOT FB_FileClose_Indo.bBusy AND NOT FB_FileClose_Indo.bError THEN FB_FileOpen_Indo.bExecute:=FALSE; IndoReport:=IndoReport+1;END_IF(*ProductionData_IndoPrint:='';*)

9:	FB_FileClose_Indo.bExecute:=FALSE;
	IF (*CycleComplete OR CycleComplete1*)ReportSave OR testbit THEN

	FB_FileOpen_Indo.bExecute:=TRUE;
	IF NOT FB_FileOpen_Indo.bBusy AND NOT FB_FileOpen_Indo.bError AND FB_FileOpen_Indo.hFile>0 THEN  ReportBot1_Indo:=TRUE;END_IF

	IF ReportBot1_Indo THEN IndoReport:=IndoReport+1;END_IF END_IF

10:
ProductionData_IndoPrint2:= CONCAT(ProductionData_IndoPrint11.S_NO,',');
ProductionData_IndoPrint2:=	 CONCAT( ProductionData_IndoPrint2,ProductionData_IndoPrint11.S_DATE	);
ProductionData_IndoPrint2:= CONCAT( ProductionData_IndoPrint2,',');
(*ProductionData_IndoPrint2:=	 CONCAT( ProductionData_IndoPrint2,ProductionData_IndoPrint11.STIME);
ProductionData_IndoPrint2:= CONCAT( ProductionData_IndoPrint2,',');*)
ProductionData_IndoPrint2:=	 CONCAT( ProductionData_IndoPrint2,ProductionData_IndoPrint11.CONETYPE	);
ProductionData_IndoPrint2:= CONCAT( ProductionData_IndoPrint2,',');
ProductionData_IndoPrint2:=	 CONCAT( ProductionData_IndoPrint2,ProductionData_IndoPrint11.CARTONNO);
ProductionData_IndoPrint2:= CONCAT( ProductionData_IndoPrint2,',');
ProductionData_IndoPrint2:=	 CONCAT( ProductionData_IndoPrint2,ProductionData_IndoPrint11.LOTNO);
ProductionData_IndoPrint2:= CONCAT( ProductionData_IndoPrint2,',');
ProductionData_IndoPrint2:=	 CONCAT( ProductionData_IndoPrint2,ProductionData_IndoPrint11.NETWT);
ProductionData_IndoPrint2:= CONCAT( ProductionData_IndoPrint2,',');
ProductionData_IndoPrint2:=	 CONCAT( ProductionData_IndoPrint2,ProductionData_IndoPrint11.WORKORDERNO);
ProductionData_IndoPrint2:= CONCAT( ProductionData_IndoPrint2,',');

ProductionData_IndoPrint2:=	 CONCAT( ProductionData_IndoPrint2,ProductionData_IndoPrint11.DFLTNTWT);
ProductionData_IndoPrint2:= CONCAT( ProductionData_IndoPrint2,',');
ProductionData_IndoPrint2:=	 CONCAT( ProductionData_IndoPrint2,ProductionData_IndoPrint11.DFLTGRSWT);
ProductionData_IndoPrint2:= CONCAT( ProductionData_IndoPrint2,',');
ProductionData_IndoPrint2:=	 CONCAT( ProductionData_IndoPrint2,ProductionData_IndoPrint11.BLEND);
ProductionData_IndoPrint2:= CONCAT( ProductionData_IndoPrint2,',');
ProductionData_IndoPrint2:=	 CONCAT( ProductionData_IndoPrint2,ProductionData_IndoPrint11.SHADE);
ProductionData_IndoPrint2:= CONCAT( ProductionData_IndoPrint2,',');
ProductionData_IndoPrint2:=	 CONCAT( ProductionData_IndoPrint2,ProductionData_IndoPrint11.CONETIP);
ProductionData_IndoPrint2:= CONCAT( ProductionData_IndoPrint2,',');
ProductionData_IndoPrint2:=	 CONCAT( ProductionData_IndoPrint2,ProductionData_IndoPrint11.CONENTWT);
ProductionData_IndoPrint2:= CONCAT( ProductionData_IndoPrint2,',');
ProductionData_IndoPrint2:=	 CONCAT( ProductionData_IndoPrint2,ProductionData_IndoPrint11.CONELENGTH);
ProductionData_IndoPrint2:= CONCAT( ProductionData_IndoPrint2,',');
ProductionData_IndoPrint2:=	 CONCAT( ProductionData_IndoPrint2,ProductionData_IndoPrint11.DOMEXP);
ProductionData_IndoPrint2:= CONCAT( ProductionData_IndoPrint2,',');
ProductionData_IndoPrint2:=	 CONCAT( ProductionData_IndoPrint2,ProductionData_IndoPrint11.PACKTYPE);
ProductionData_IndoPrint2:= CONCAT( ProductionData_IndoPrint2,',');
ProductionData_IndoPrint2:=	 CONCAT( ProductionData_IndoPrint2,ProductionData_IndoPrint11.COUNTCODE);
ProductionData_IndoPrint2:= CONCAT( ProductionData_IndoPrint2,'$0A');
(*ProductionData_IndoPrint2:=	 CONCAT( ProductionData_IndoPrint2,ProductionData_IndoPrint11.DFLTGROSSWEIGHT);
ProductionData_IndoPrint2:= CONCAT( ProductionData_IndoPrint2,',');
ProductionData_IndoPrint2:=	 CONCAT( ProductionData_IndoPrint2,ProductionData_IndoPrint11.ACTGROSSWEIGHT);
ProductionData_IndoPrint2:= CONCAT( ProductionData_IndoPrint2,'$0A');
ProductionData_IndoPrint2:=	 CONCAT( ProductionData_IndoPrint2,ProductionData_IndoPrint11.NetWt9);
ProductionData_IndoPrint2:= CONCAT( ProductionData_IndoPrint2,',');
ProductionData_IndoPrint2:=	 CONCAT( ProductionData_IndoPrint2,ProductionData_IndoPrint11.NetWt10);
ProductionData_IndoPrint2:= CONCAT( ProductionData_IndoPrint2,',');
ProductionData_IndoPrint2:=	 CONCAT( ProductionData_IndoPrint2,ProductionData_IndoPrint11.NetWt11);
ProductionData_IndoPrint2:= CONCAT( ProductionData_IndoPrint2,',');
ProductionData_IndoPrint2:=	 CONCAT( ProductionData_IndoPrint2,ProductionData_IndoPrint11.NetWt12);
ProductionData_IndoPrint2:= CONCAT( ProductionData_IndoPrint2,',');*)
ReportBot1_Indo:=FALSE;ReportSave:=FALSE;CycleComplete:=FALSE;CycleComplete1:=FALSE;testbit:=FALSE;
IndoReport:=15;


11:	ProductionDataValues_IndoPrint_Com:=ProductionData_IndoPrint2;
TON_Indo3(IN:=TRUE , PT:=t#5s , Q=> , ET=> );
	FB_FileWrite_Indo.bExecute:=TRUE;
	IF NOT FB_FileWrite_Indo.bBusy AND NOT FB_FileWrite_Indo.bError AND TON_Indo3.Q THEN IndoReport:=IndoReport+1; END_IF

12:	FB_FileWrite_Indo.bExecute:=FALSE;(*ProductionData_IndoPrint:='';*)IndoReport:=IndoReport+1;

13:	ReportBot2_Indo:=TRUE;
	IF ReportBot2_Indo THEN IndoReport:=IndoReport+1;END_IF

14:(*	ProductionData_IndoPrint2:= CONCAT(ProductionData_IndoPrint11.NetWt13,',');
ProductionData_IndoPrint2:=	 CONCAT( ProductionData_IndoPrint2,ProductionData_IndoPrint11.NetWt14	);
ProductionData_IndoPrint2:= CONCAT( ProductionData_IndoPrint2,',');
ProductionData_IndoPrint2:=	 CONCAT( ProductionData_IndoPrint2,ProductionData_IndoPrint11.NetWt15);
ProductionData_IndoPrint2:= CONCAT( ProductionData_IndoPrint2,',');
ProductionData_IndoPrint2:=	 CONCAT( ProductionData_IndoPrint2,ProductionData_IndoPrint11.NetWt16);
ProductionData_IndoPrint2:= CONCAT( ProductionData_IndoPrint2,',');
ProductionData_IndoPrint2:=	 CONCAT( ProductionData_IndoPrint2,ProductionData_IndoPrint11.NetWt17);
ProductionData_IndoPrint2:= CONCAT( ProductionData_IndoPrint2,',');
ProductionData_IndoPrint2:=	 CONCAT( ProductionData_IndoPrint2,ProductionData_IndoPrint11.NetWt18);
ProductionData_IndoPrint2:= CONCAT( ProductionData_IndoPrint2,',');
ProductionData_IndoPrint2:=	 CONCAT( ProductionData_IndoPrint2,ProductionData_IndoPrint11.NetWt19);
ProductionData_IndoPrint2:= CONCAT( ProductionData_IndoPrint2,',');
ProductionData_IndoPrint2:=	 CONCAT( ProductionData_IndoPrint2,ProductionData_IndoPrint11.NetWt20);
ProductionData_IndoPrint2:= CONCAT( ProductionData_IndoPrint2,',');
ProductionData_IndoPrint2:=	 CONCAT( ProductionData_IndoPrint2,ProductionData_IndoPrint11.NetWt21);
ProductionData_IndoPrint2:= CONCAT( ProductionData_IndoPrint2,',');
ProductionData_IndoPrint2:=	 CONCAT( ProductionData_IndoPrint2,ProductionData_IndoPrint11.NetWt22);
ProductionData_IndoPrint2:= CONCAT( ProductionData_IndoPrint2,',');
ProductionData_IndoPrint2:=	 CONCAT( ProductionData_IndoPrint2,ProductionData_IndoPrint11.NetWt23);
ProductionData_IndoPrint2:= CONCAT( ProductionData_IndoPrint2,',');
ProductionData_IndoPrint2:=	 CONCAT( ProductionData_IndoPrint2,ProductionData_IndoPrint11.NetWt24);
ProductionData_IndoPrint2:= CONCAT( ProductionData_IndoPrint2,'$0A');*)
ReportBot2_Indo:=FALSE;
IndoReport:=IndoReport+1;

15:ProductionDataValues_IndoPrint_Com:=ProductionData_IndoPrint2;
TON_Indo4(IN:=TRUE , PT:=t#5s , Q=> , ET=> );

	FB_FileWrite_Indo.bExecute:=TRUE; IndoReport:=IndoReport+1;
	(*IF NOT FB_FileWrite_Indo.bBusy AND NOT FB_FileWrite_Indo.bError AND TON_Indo4.Q  THEN IndoReport:=IndoReport+1;END_IF*)

16:	IF NOT FB_FileWrite_Indo.bBusy AND NOT FB_FileWrite_Indo.bError THEN FB_FileWrite_Indo.bExecute:=FALSE; IndoReport:=IndoReport+1;END_IF


17:	TON_Indo3(IN:=FALSE);TON_Indo4(IN:=FALSE);TON_Indo2(IN:=FALSE);TON_Indo1(IN:=FALSE);FB_FileWrite_Indo.bExecute:=FALSE;PrintOk:=TRUE;IndoReport:=IndoReport+1;

18:	FB_FileClose_Indo.bExecute:=TRUE;
	 IF NOT FB_FileClose_Indo.bBusy AND NOT FB_FileClose_Indo.bError THEN  IndoReport:=20;END_IF

19:	IF bANewDay THEN IndoReport:=IndoReport+1;
	ELSIF NOT bANewDay THEN FB_FileOpen_Indo.bExecute:=FALSE; IndoReport:=9;
END_IF

20:	FB_FileOpen_Indo.bExecute:=FALSE;SerialNo:=SerialNo+1;BagSerialNo:=BagSerialNo+1;IndoReport:=9;

END_CASE



IF sDay <> sOldDay THEN bANewDay:=TRUE;IndoReport:=0; END_IF
TON_NEWDAY(IN:=bANewDay , PT:=T#0.5s , Q=> , ET=> );




CASE WriteError OF

0:	IF FB_FileWrite_Indo.bError THEN FB_FileWrite_Indo.bExecute:=FALSE;TON_writedly(IN:=FALSE);
	WriteError:=WriteError+1;END_IF

1:	TON_writedly(IN:=TRUE , PT:=t#2s , Q=> , ET=> );
	IF TON_writedly.Q THEN FB_FileWrite_Indo.bExecute:=TRUE;WriteError:=WriteError+1;END_IF

2:	TON_writedly(IN:=FALSE);WriteError:=0;

END_CASE




CASE OpenError OF

0:	IF FB_FileOpen_Indo.bError THEN FB_FileOpen_Indo.bExecute:=FALSE;TON_Opendly(IN:=FALSE);
	OpenError:=OpenError+1;END_IF

1:	TON_Opendly(IN:=TRUE , PT:=t#2s , Q=> , ET=> );
	IF TON_Opendly.Q THEN FB_FileOpen_Indo.bExecute:=TRUE;OpenError:=OpenError+1;END_IF

2:	TON_Opendly(IN:=FALSE);OpenError:=0;

END_CASE










		ProductionData_IndoPrint11.S_NO	:=DINT_TO_STRING(SerialNo);
		ProductionData_IndoPrint11.S_DATE	:=(sDATEFinal);
		ProductionData_IndoPrint11.CONETYPE	:=INT_TO_STRING( iATotalNoOfCones );
		ProductionData_IndoPrint11.CARTONNO	:=DINT_TO_STRING(CARTONNO_DIS);
		ProductionData_IndoPrint11.LOTNO	:=(LOTNO_DIS);
		ProductionData_IndoPrint11.NETWT	:=REAL_TO_STRING(var_5);
		ProductionData_IndoPrint11.WORKORDERNO	:=(WORKORDERNO_DIS);
		ProductionData_IndoPrint11.DFLTNTWT	:=REAL_TO_STRING (DFLTNETWT_DIS);
		ProductionData_IndoPrint11.DFLTGRSWT	:=REAL_TO_STRING(DFLTGROSSWT_DIS);
		ProductionData_IndoPrint11.BLEND	:=(BLEND_DIS);
		ProductionData_IndoPrint11.SHADE	:=(SHADE_DIS );
		ProductionData_IndoPrint11.CONETIP	:=(CONETIP_DIS);
		ProductionData_IndoPrint11.CONENTWT	:=REAL_TO_STRING(CONENETWT_DIS);
		ProductionData_IndoPrint11.CONELENGTH	:=REAL_TO_STRING (CONELENGTH_DIS);
		ProductionData_IndoPrint11.DOMEXP	:=(DOM_EXPORT_DIS);
		ProductionData_IndoPrint11.PACKTYPE	:=(PACKTYPE_DIS);
		ProductionData_IndoPrint11.COUNTCODE	:=(COUNT_DIS);
(*
		ProductionData_IndoPrint11.NetWt17	:=REAL_TO_STRING(Cone_17_Wt);
		ProductionData_IndoPrint11.NetWt18	:=REAL_TO_STRING(Cone_18_Wt);
		ProductionData_IndoPrint11.NetWt19	:=REAL_TO_STRING(Cone_19_Wt);
		ProductionData_IndoPrint11.NetWt20	:=REAL_TO_STRING(Cone_20_Wt);
		ProductionData_IndoPrint11.NetWt21	:=REAL_TO_STRING(Cone_21_Wt);
		ProductionData_IndoPrint11.NetWt22	:=REAL_TO_STRING(Cone_22_Wt);
		ProductionData_IndoPrint11.NetWt23	:=REAL_TO_STRING(Cone_23_Wt);
		ProductionData_IndoPrint11.NetWt24	:=REAL_TO_STRING(Cone_24_Wt);

		stStation1_ProductionData.S_No						:=INT_TO_STRING( Pgm_NoHmi );
		stStation1_ProductionData.ConeType				:=INT_TO_STRING( iATotalNoOfCones );
		stStation1_ProductionData.CartonNo					:=INT_TO_STRING(CurrentCartonNo)(*CartonNoHmi*);
		stStation1_ProductionData.LotNo					:= (iLotNoHmi);
		stStation1_ProductionData.SDateF					:= (sDATEFinal);
		stStation1_ProductionData.NetWt					:=REAL_TO_STRING(var_5);
		stStation1_ProductionData.WorkOrderNo				:= (iWorkOrderNoHmi);
		stStation1_ProductionData.DefaultNettWeight			:=REAL_TO_STRING (DefaultNetWeightHmi);
		stStation1_ProductionData.DefaultGrossWeight		:= REAL_TO_STRING(DefaultGrossWeightHmi);
		stStation1_ProductionData.Blend					:= (BlendHmi);
		stStation1_ProductionData.Shade					:= (ShadeHmi );
		stStation1_ProductionData.ConeTip					:= (ConeTipHmi);
		stStation1_ProductionData.ConeNettWeight			:= (*REAL_TO_STRING*)(ConeNettHmi);
		stStation1_ProductionData.ConeLength				:=REAL_TO_STRING (ConeLengthHmi);
		stStation1_ProductionData.Dom_Exp					:= (Dom_ExpHmi);
		stStation1_ProductionData.PackType				:= (PackTypeHmi);
		stStation1_ProductionData.CountCode				:= (CountCodeHmi);


*)

*)
END_PROGRAM

(* POU AutoMode/DATAERRORLOG_REPORT, ST *)
PROGRAM DATAERRORLOG_REPORT
VAR
	FB_FileOpen_Indo: FB_FileOpen;
	FB_FileWrite_Indo: FB_FileWrite;
	FB_FileClose_Indo: FB_FileClose;
	FB_FileDelete_Indo: FB_FileDelete;
	R_TRIG_ERROR1: R_TRIG;
	ERROR1: BOOL;
	ERROR1DIS: STRING;

	R_TRIG_ERROR2: R_TRIG;
	ERROR2: BOOL;
	ERROR2DIS: STRING;

	R_TRIG_ERROR3: R_TRIG;
	ERROR3: BOOL;
	ERROR3DIS: STRING;
	AlarmData: STRING;
	R_TRIG_IndoPrintError: R_TRIG;
	TON_NEWDAYError: TON;
	TON_NewdaydlyError: TON;
	bANewDayError: BOOL;

	ReportHead1Error_Indo: BOOL;
	bANewDayErrror: BOOL;
	ReportHead1Errror_Indo: BOOL;
	TON_Indo2: TON;
	ReportBot1Error_Indo: BOOL;
	TON_Indo3: TON;
	IndoReport: INT;
	ReportBot2Error_Indo: BOOL;
	ReportSaveErrror: BOOL;
	ReportSaveError: BOOL;
	testbit: BOOL;
	sOldDayError: STRING;
	TON_Newdaydly: TON;
	TON_Indo1: TON;
	ReportHead2Error_Indo: BOOL;
	TON_Indo4: TON;
	R_TRIG_ErrorRepo: R_TRIG;
	ERROR_Report: BOOL;
	STEPERROR: INT;
	WriteError: INT;
	TON_writedly: TON;
	OpenError: INT;
	TON_Opendly: TON;
	R_TRIG_ErrorRepo_Int: R_TRIG;
END_VAR
IF bAConeFeedCylRsError OR   bPloySheetSensError OR bAFwdCylRsError OR bAWrappingCylRsError OR bASupplyPressureError OR
bAPolythinSheetError OR  ConeAlignErr OR bASealTopBotCylRsError OR bASealSepXCylRsError OR bASealSepYCylRsError
 OR bAConeMissAtSealConv  OR bAEmergencyPressed OR bCheckWrappingSen  OR
 bCheckWrappingSen2 OR bCheckWrappingSen3  OR bGrossWieghtNOk  OR bGrossWtCylEndSenError
 THEN ERROR_Report:=TRUE;
END_IF

IF bAConeFeedCylRsError THEN AlarmData:='CONE FEEDING PISTON END READ SWITCH ERROR';END_IF

IF bAFwdCylRsError THEN AlarmData:='ONE FORWARD PISTON  END READ SWITCH ERROR';END_IF

IF bAWrappingCylRsError THEN AlarmData:='WRAPPING  PISTON  END READ SWITCH ERROR';END_IF


IF bASealTopBotCylRsError THEN AlarmData:='SEALING TOP PISTON  END READ SWITCH ERROR';END_IF

IF bASealSepXCylRsError THEN AlarmData:='SEALING X AXIS PISTON  END READ SWITCH ERROR';END_IF

IF bGrossWieghtNOk THEN AlarmData:='GROSS WEIGHT NOT OK';END_IF

IF bGrossWtCylEndSenError THEN AlarmData:='GROSS WEIGHT PISTON  END READ SWITCH ERROR';END_IF

IF bAConeMissAtSealConv THEN AlarmData:='CONE MISS IN SEALING CONVEYOR';END_IF

IF bAEmergencyPressed THEN AlarmData:='EMERGENCY PRESSED';END_IF

IF bASealSepYCylRsError THEN AlarmData:='Y AXIS PISTON END READ SWITCH ERROR';END_IF

IF bPloySheetSensError OR bAPolythinSheetError THEN AlarmData:='POLYTHENE SHEET NOT FEED ERROR';END_IF

IF bASupplyPressureError THEN AlarmData:='SUPPLY PRESSURE ERROR';END_IF

IF ConeAlignErr THEN AlarmData:='WRAP CONE ALAIGN ERROR';END_IF

IF R_TRIG_ErrorRepo_Int.Q THEN  AlarmData:='MACHINE INITIALIZE STARTED';END_IF

FB_FileOpen_Indo(
	sNetId:='192.168.225.201.1.1',
	sPathName:= ReportPath_Final_2Error,
	nMode:=FOPEN_MODEAPPEND ,
	ePath:=PATH_GENERIC ,
	bExecute:= ,
	tTimeout:=T#2s ,
	bBusy=> ,
	bError=> ,
	nErrId=> ,
	hFile=> );

FB_FileWrite_Indo(
	sNetId:='192.168.225.201.1.1',
	hFile:=FB_FileOpen_Indo.hFile ,
	pWriteBuff:=ADR(ProductionDataValuesError_IndoPrint_Com),
	cbWriteLen:=LEN(ProductionDataValuesError_IndoPrint_Com),
	bExecute:= ,
	tTimeout:=T#2s ,
	bBusy=> ,
	bError=> ,
	nErrId=> ,
	cbWrite=> );


FB_FileClose_Indo(
	sNetId:='192.168.225.201.1.1',
	hFile:=FB_FileOpen_Indo.hFile ,
	bExecute:= ,
	tTimeout:=T#2s ,
	bBusy=> ,
	bError=> ,
	nErrId=> );

FB_FileDelete_Indo(
	sNetId:='192.168.225.201.1.1',
	sPathName:= ReportPath_Final_2Error,
	ePath:=PATH_GENERIC ,
	bExecute:= ,
	tTimeout:=T#2s ,
	bBusy=> ,
	bError=> ,
	nErrId=> );


CASE STEPERROR OF
0:IF FB_FileOpen_Indo.bError THEN FB_FileOpen_Indo.bExecute:=FALSE;STEPERROR:=STEPERROR+1;END_IF

1:FB_FileOpen_Indo.bExecute:=TRUE;STEPERROR:=STEPERROR+1;


2:IF NOT FB_FileOpen_Indo.bError THEN STEPERROR:=0;END_IF

END_CASE

R_TRIG_IndoPrintError(CLK:=( bANewDayError )  , Q=> );

R_TRIG_ErrorRepo(CLK:=bAError , Q=> );



CASE IndoReport OF
0:	  IF TON_NEWDAYError.Q   THEN	sOldDayError := sDay;TON_NewdaydlyError(IN:=TRUE , PT:=t#0.2s , Q=> , ET=> );
		IF TON_NewdaydlyError.Q THEN
		bANewDayError:=FALSE;TON_NewdaydlyError(IN:=FALSE);TON_NEWDAYError(IN:=FALSE);IndoReport:=1; SerialNoError:=1;
		FB_FileOpen_Indo.bExecute:=TRUE;END_IF END_IF

1:	TON_NewdaydlyError(IN:=FALSE);bANewDay:=FALSE;
	IF NOT FB_FileOpen_Indo.bBusy AND NOT FB_FileOpen_Indo.bError AND FB_FileOpen_Indo.hFile>0 THEN ReportHead1Error_Indo:=TRUE;END_IF

	IF ReportHead1Error_Indo THEN
	ProductionDataError_IndoPrint:= CONCAT( 'SL NO',',');
	ProductionDataError_IndoPrint:=	 CONCAT( ProductionDataError_IndoPrint,'TIME');
		ProductionDataError_IndoPrint:= CONCAT( ProductionDataError_IndoPrint,',');
	(*ProductionDataError_IndoPrint:=	 CONCAT( ProductionDataError_IndoPrint,'TIME');
		ProductionDataError_IndoPrint:=CONCAT( ProductionDataError_IndoPrint,',');
	ProductionDataError_IndoPrint:=	 CONCAT( ProductionDataError_IndoPrint,'SHIFT');
		ProductionDataError_IndoPrint:= CONCAT( ProductionDataError_IndoPrint,',');*)
	ProductionDataError_IndoPrint:=	 CONCAT( ProductionDataError_IndoPrint,'ERROR');
		ProductionDataError_IndoPrint:= CONCAT( ProductionDataError_IndoPrint,'$0A');
	(*ProductionDataError_IndoPrint:=	 CONCAT( ProductionData_IndoPrint,'LOT NO');
		ProductionDataError_IndoPrint:=CONCAT( ProductionData_IndoPrint,',');
	ProductionDataError_IndoPrint:=	 CONCAT( ProductionData_IndoPrint,'DFLT NET WT');
		ProductionDataError_IndoPrint:=CONCAT( ProductionData_IndoPrint,',');
	ProductionDataError_IndoPrint:=	 CONCAT( ProductionData_IndoPrint,'ACT NET WT');
		ProductionDataError_IndoPrint:= CONCAT( ProductionData_IndoPrint,'$0A');
ProductionData_IndoPrint:=	 CONCAT( ProductionData_IndoPrint,'DFLT GROSS WT');
		ProductionData_IndoPrint:=CONCAT( ProductionData_IndoPrint,',');
ProductionData_IndoPrint:=	 CONCAT( ProductionData_IndoPrint,'ACT GROSS WT');
		ProductionData_IndoPrint:= CONCAT( ProductionData_IndoPrint,'$0A');
ProductionData_IndoPrint:=	 CONCAT( ProductionData_IndoPrint,'Cn9Wt');
		ProductionData_IndoPrint:=CONCAT( ProductionData_IndoPrint,',');
ProductionData_IndoPrint:=	 CONCAT( ProductionData_IndoPrint,'Cn10Wt');
		ProductionData_IndoPrint:=CONCAT( ProductionData_IndoPrint,',');
ProductionData_IndoPrint:=	 CONCAT( ProductionData_IndoPrint,'Cn11Wt');
		ProductionData_IndoPrint:=CONCAT( ProductionData_IndoPrint,',');
ProductionData_IndoPrint:=	 CONCAT( ProductionData_IndoPrint,'Cn12Wt');
	ProductionData_IndoPrint:=CONCAT( ProductionData_IndoPrint,',');*)
IndoReport:=7; END_IF

2:	PROCESSCOMPLETE:=FALSE;ReportHead1Error_Indo:=FALSE;ProductionDataValuesError_IndoPrint_Com:=ProductionDataError_IndoPrint;
	TON_Indo1(IN:=TRUE , PT:=t#5s , Q=> , ET=> );
	FB_FileWrite_Indo.bExecute:=TRUE;
	IF NOT FB_FileWrite_Indo.bBusy AND NOT FB_FileWrite_Indo.bError AND FB_FileWrite_Indo.hFile>0 AND TON_Indo1.Q THEN IndoReport:=IndoReport+1; END_IF

3:	ProductionDataValues_IndoPrint_Com:=ProductionData_IndoPrint;
	FB_FileWrite_Indo.bExecute:=TRUE;
	IF NOT FB_FileWrite_Indo.bBusy AND NOT FB_FileWrite_Indo.bError THEN IndoReport:=IndoReport+1; END_IF

4:	FB_FileWrite_Indo.bExecute:=FALSE;ProductionData_IndoPrint:='';IndoReport:=IndoReport+1;

5:	ReportHead2Error_Indo:=TRUE;
	IF ReportHead2Error_Indo THEN IndoReport:=IndoReport+1;END_IF

6:	ProductionData_IndoPrint:=	 CONCAT( ProductionData_IndoPrint,'Cn13Wt');
		ProductionData_IndoPrint:=CONCAT( ProductionData_IndoPrint,',');
ProductionData_IndoPrint:=	 CONCAT( ProductionData_IndoPrint,'Cn14Wt');
		ProductionData_IndoPrint:=CONCAT( ProductionData_IndoPrint,',');
ProductionData_IndoPrint:=	 CONCAT( ProductionData_IndoPrint,'Cn15Wt');
		ProductionData_IndoPrint:=CONCAT( ProductionData_IndoPrint,',');
ProductionData_IndoPrint:=	 CONCAT( ProductionData_IndoPrint,'Cn16Wt');
		ProductionData_IndoPrint:=CONCAT( ProductionData_IndoPrint,',');
ProductionData_IndoPrint:=	 CONCAT( ProductionData_IndoPrint,'Cn17Wt');
		ProductionData_IndoPrint:=CONCAT( ProductionData_IndoPrint,',');
ProductionData_IndoPrint:=	 CONCAT( ProductionData_IndoPrint,'Cn18Wt');
		ProductionData_IndoPrint:=CONCAT( ProductionData_IndoPrint,',');
ProductionData_IndoPrint:=	 CONCAT( ProductionData_IndoPrint,'Cn19Wt');
		ProductionData_IndoPrint:=CONCAT( ProductionData_IndoPrint,',');
ProductionData_IndoPrint:=	 CONCAT( ProductionData_IndoPrint,'Cn20Wt');
		ProductionData_IndoPrint:=CONCAT( ProductionData_IndoPrint,',');
ProductionData_IndoPrint:=	 CONCAT( ProductionData_IndoPrint,'Cn21Wt');
		ProductionData_IndoPrint:=CONCAT( ProductionData_IndoPrint,',');
ProductionData_IndoPrint:=	 CONCAT( ProductionData_IndoPrint,'Cn22Wt');
		ProductionData_IndoPrint:=CONCAT( ProductionData_IndoPrint,',');
ProductionData_IndoPrint:=	 CONCAT( ProductionData_IndoPrint,'Cn23Wt');
		ProductionData_IndoPrint:=CONCAT( ProductionData_IndoPrint,',');
	ProductionData_IndoPrint:=	 CONCAT( ProductionData_IndoPrint,'Cn24Wt');
ProductionData_IndoPrint:= CONCAT( ProductionData_IndoPrint,'$0A');
ReportHead2Error_Indo:=FALSE;
IndoReport:=IndoReport+1;

7:	ReportHead1Error_Indo:=FALSE;ProductionDataValuesError_IndoPrint_Com:=ProductionDataError_IndoPrint;
TON_Indo2(IN:=TRUE , PT:=t#5s , Q=> , ET=> );
	FB_FileWrite_Indo.bExecute:=TRUE;
	IF NOT FB_FileWrite_Indo.bBusy AND NOT FB_FileWrite_Indo.bError  AND TON_Indo2.Q THEN  IndoReport:=IndoReport+1; END_IF

8:	FB_FileWrite_Indo.bExecute:=FALSE;
	FB_FileClose_Indo.bExecute:=TRUE;
	 IF NOT FB_FileClose_Indo.bBusy AND NOT FB_FileClose_Indo.bError THEN FB_FileOpen_Indo.bExecute:=FALSE; IndoReport:=IndoReport+1;END_IF(*ProductionData_IndoPrint:='';*)

9:	FB_FileClose_Indo.bExecute:=FALSE;
	IF R_TRIG_ErrorRepo.Q OR R_TRIG_ErrorRepo_Int.Q OR testbit THEN

	FB_FileOpen_Indo.bExecute:=TRUE;
	IF NOT FB_FileOpen_Indo.bBusy AND NOT FB_FileOpen_Indo.bError AND FB_FileOpen_Indo.hFile>0 THEN  ReportBot1Error_Indo:=TRUE;END_IF

	IF ReportBot1Error_Indo THEN IndoReport:=IndoReport+1;END_IF END_IF

